LIN {X -0.215,Y -608.522,Z 1231.656,A 0.000,B 0.000,C 90.000,E1 154.152} C_DIS
LIN {X 0.197,Y -611.712,Z 1231.652,A 0.000,B 0.000,C 90.000,E1 153.332} C_DIS
LIN {X 0.064,Y -615.753,Z 1231.646,A 0.000,B 0.000,C 90.000,E1 152.308} C_DIS
LIN {X -0.293,Y -621.493,Z 1231.638,A 0.000,B 0.000,C 90.000,E1 150.795} C_DIS
LIN {X -0.001,Y -625.230,Z 1231.632,A 0.000,B 0.000,C 90.000,E1 149.744} C_DIS
LIN {X -0.198,Y -628.990,Z 1231.626,A 0.000,B 0.000,C 90.000,E1 148.742} C_DIS
LIN {X 0.009,Y -633.541,Z 1231.619,A 0.000,B 0.000,C 90.000,E1 147.454} C_DIS
LIN {X -0.240,Y -637.777,Z 1231.612,A 0.000,B 0.000,C 90.000,E1 146.215} C_DIS
LIN {X -0.421,Y -641.797,Z 1231.605,A 0.000,B 0.000,C 90.000,E1 144.975} C_DIS
LIN {X -0.172,Y -645.344,Z 1231.598,A 0.000,B 0.000,C 90.000,E1 143.703} C_DIS
LIN {X -0.235,Y -646.733,Z 1231.596,A 0.000,B 0.000,C 90.000,E1 143.210} C_DIS
LIN {X -0.024,Y -649.852,Z 1231.589,A 0.000,B 0.000,C 90.000,E1 141.949} C_DIS
LIN {X 0.287,Y -653.430,Z 1231.580,A 0.000,B 0.000,C 90.000,E1 140.436} C_DIS
LIN {X 0.118,Y -656.246,Z 1231.573,A 0.000,B 0.000,C 90.000,E1 139.218} C_DIS
LIN {X -0.055,Y -660.199,Z 1231.564,A 0.000,B 0.000,C 90.000,E1 137.514} C_DIS
LIN {X -0.154,Y -664.675,Z 1231.553,A 0.000,B 0.000,C 90.000,E1 135.567} C_DIS
LIN {X -0.165,Y -668.917,Z 1231.544,A 0.000,B 0.000,C 90.000,E1 133.866} C_DIS
LIN {X -0.055,Y -673.267,Z 1231.534,A 0.000,B 0.000,C 90.000,E1 132.162} C_DIS
LIN {X 0.130,Y -676.933,Z 1231.526,A 0.000,B 0.000,C 90.000,E1 130.701} C_DIS
LIN {X -0.089,Y -680.001,Z 1231.520,A 0.000,B 0.000,C 90.000,E1 129.519} C_DIS
LIN {X -0.223,Y -683.658,Z 1231.512,A 0.000,B 0.000,C 90.000,E1 128.096} C_DIS
LIN {X -0.178,Y -687.277,Z 1231.504,A 0.000,B 0.000,C 90.000,E1 126.664} C_DIS
LIN {X -0.296,Y -689.544,Z 1231.498,A 0.000,B 0.000,C 90.000,E1 125.724} C_DIS
LIN {X 0.024,Y -692.770,Z 1231.490,A 0.000,B 0.000,C 90.000,E1 124.278} C_DIS
LIN {X 0.183,Y -695.394,Z 1231.484,A 0.000,B 0.000,C 90.000,E1 123.086} C_DIS
LIN {X 0.339,Y -697.341,Z 1231.479,A 0.000,B 0.000,C 90.000,E1 122.133} C_DIS
LIN {X -0.187,Y -699.644,Z 1231.472,A 0.000,B 0.000,C 90.000,E1 121.003} C_DIS
LIN {X 0.015,Y -701.391,Z 1231.467,A 0.000,B 0.000,C 90.000,E1 120.050} C_DIS
LIN {X -0.121,Y -703.044,Z 1231.462,A 0.000,B 0.000,C 90.000,E1 119.127} C_DIS
LIN {X 0.099,Y -704.093,Z 1231.458,A 0.000,B 0.000,C 90.000,E1 118.409} C_DIS
LIN {X 0.000,Y -704.953,Z 1231.454,A 0.000,B 0.000,C 90.000,E1 117.719} C_DIS
LIN {X 0.241,Y -705.565,Z 1231.450,A 0.000,B 0.000,C 90.000,E1 117.001} C_DIS
LIN {X 0.170,Y -706.015,Z 1231.446,A 0.000,B 0.000,C 90.000,E1 116.309} C_DIS
LIN {X 0.413,Y -706.169,Z 1231.442,A 0.000,B 0.000,C 90.000,E1 115.591} C_DIS
LIN {X 0.058,Y -706.120,Z 1231.440,A 0.000,B 0.000,C 90.000,E1 115.155} C_DIS
LIN {X 0.001,Y -705.807,Z 1231.437,A 0.000,B 0.000,C 90.000,E1 114.695} C_DIS
LIN {X -0.003,Y -705.533,Z 1231.436,A 0.000,B 0.000,C 90.000,E1 114.463} C_DIS
LIN {X -0.069,Y -704.719,Z 1231.433,A 0.000,B 0.000,C 90.000,E1 114.003} C_DIS
LIN {X -0.069,Y -703.824,Z 1231.432,A 0.000,B 0.000,C 90.000,E1 113.770} C_DIS
LIN {X -0.429,Y -701.590,Z 1231.429,A 0.000,B 0.000,C 90.000,E1 113.334} C_DIS
LIN {X -0.291,Y -700.673,Z 1231.429,A 0.000,B 0.000,C 90.000,E1 113.206} C_DIS
LIN {X 0.148,Y -695.709,Z 1231.426,A 0.000,B 0.000,C 90.000,E1 112.717} C_DIS
LIN {X -0.315,Y -694.073,Z 1231.426,A 0.000,B 0.000,C 90.000,E1 112.642} C_DIS
LIN {X 0.049,Y -691.649,Z 1231.425,A 0.000,B 0.000,C 90.000,E1 112.514} C_DIS
LIN {X -0.259,Y -686.935,Z 1231.424,A 0.000,B 0.000,C 90.000,E1 112.386} C_DIS
LIN {X -0.290,Y -683.690,Z 1231.424,A 0.000,B 0.000,C 90.000,E1 112.333} C_DIS
LIN {X -0.124,Y -676.958,Z 1231.424,A 0.000,B 0.000,C 90.000,E1 112.280} C_DIS
LIN {X -0.162,Y -617.564,Z 1231.424,A 0.000,B 0.000,C 90.000,E1 112.280} C_DIS
LIN {X 0.169,Y -614.890,Z 1231.423,A 0.000,B 0.000,C 90.000,E1 112.099} C_DIS
LIN {X -0.080,Y -611.777,Z 1231.421,A 0.000,B 0.000,C 90.000,E1 111.844} C_DIS
LIN {X 0.070,Y -611.245,Z 1231.421,A 0.000,B 0.000,C 90.000,E1 111.770} C_DIS
LIN {X -0.103,Y -610.878,Z 1231.421,A 0.000,B 0.000,C 90.000,E1 111.716} C_DIS
LIN {X -0.008,Y -610.901,Z 1231.420,A 0.000,B 0.000,C 90.000,E1 111.535} C_DIS
LIN {X -0.055,Y -611.491,Z 1231.418,A 0.000,B 0.000,C 90.000,E1 111.280} C_DIS
LIN {X -0.324,Y -612.402,Z 1231.417,A 0.000,B 0.000,C 90.000,E1 111.046} C_DIS
LIN {X -0.008,Y -617.164,Z 1231.411,A 0.000,B 0.000,C 90.000,E1 109.993} C_DIS
LIN {X 0.052,Y -620.407,Z 1231.407,A 0.000,B 0.000,C 90.000,E1 109.214} C_DIS
LIN {X -0.211,Y -622.301,Z 1231.404,A 0.000,B 0.000,C 90.000,E1 108.725} C_DIS
LIN {X 0.129,Y -624.409,Z 1231.401,A 0.000,B 0.000,C 90.000,E1 108.181} C_DIS
LIN {X -0.348,Y -631.904,Z 1231.391,A 0.000,B 0.000,C 90.000,E1 106.441} C_DIS
LIN {X 0.056,Y -634.072,Z 1231.388,A 0.000,B 0.000,C 90.000,E1 105.898} C_DIS
LIN {X 0.126,Y -636.956,Z 1231.384,A 0.000,B 0.000,C 90.000,E1 105.134} C_DIS
LIN {X -0.226,Y -639.190,Z 1231.380,A 0.000,B 0.000,C 90.000,E1 104.411} C_DIS
LIN {X 0.061,Y -640.555,Z 1231.377,A 0.000,B 0.000,C 90.000,E1 103.883} C_DIS
LIN {X 0.045,Y -642.355,Z 1231.372,A 0.000,B 0.000,C 90.000,E1 102.883} C_DIS
LIN {X -0.111,Y -642.699,Z 1231.370,A 0.000,B 0.000,C 90.000,E1 102.647} C_DIS
LIN {X 0.206,Y -642.910,Z 1231.367,A 0.000,B 0.000,C 90.000,E1 102.119} C_DIS
LIN {X 0.240,Y -642.508,Z 1231.363,A 0.000,B 0.000,C 90.000,E1 101.366} C_DIS
LIN {X -0.072,Y -641.928,Z 1231.361,A 0.000,B 0.000,C 90.000,E1 100.894} C_DIS
LIN {X 0.238,Y -640.857,Z 1231.358,A 0.000,B 0.000,C 90.000,E1 100.366} C_DIS
LIN {X -0.202,Y -639.493,Z 1231.355,A 0.000,B 0.000,C 90.000,E1 99.905} C_DIS
LIN {X 0.088,Y -637.800,Z 1231.352,A 0.000,B 0.000,C 90.000,E1 99.378} C_DIS
LIN {X 0.263,Y -635.771,Z 1231.349,A 0.000,B 0.000,C 90.000,E1 98.859} C_DIS
LIN {X 0.080,Y -634.653,Z 1231.348,A 0.000,B 0.000,C 90.000,E1 98.624} C_DIS
LIN {X 0.091,Y -631.158,Z 1231.344,A 0.000,B 0.000,C 90.000,E1 97.992} C_DIS
LIN {X 0.224,Y -627.938,Z 1231.342,A 0.000,B 0.000,C 90.000,E1 97.473} C_DIS
LIN {X -0.134,Y -625.212,Z 1231.340,A 0.000,B 0.000,C 90.000,E1 97.125} C_DIS
LIN {X -0.123,Y -619.843,Z 1231.336,A 0.000,B 0.000,C 90.000,E1 96.486} C_DIS
LIN {X 0.026,Y -616.006,Z 1231.334,A 0.000,B 0.000,C 90.000,E1 96.087} C_DIS
LIN {X -0.273,Y -610.789,Z 1231.331,A 0.000,B 0.000,C 90.000,E1 95.625} C_DIS
LIN {X 0.251,Y -607.948,Z 1231.330,A 0.000,B 0.000,C 90.000,E1 95.334} C_DIS
LIN {X -0.273,Y -601.860,Z 1231.327,A 0.000,B 0.000,C 90.000,E1 94.935} C_DIS
LIN {X 0.266,Y -595.811,Z 1231.325,A 0.000,B 0.000,C 90.000,E1 94.473} C_DIS
LIN {X 0.137,Y -591.134,Z 1231.323,A 0.000,B 0.000,C 90.000,E1 94.188} C_DIS
LIN {X 0.120,Y -582.888,Z 1231.321,A 0.000,B 0.000,C 90.000,E1 93.726} C_DIS
LIN {X -0.057,Y -572.286,Z 1231.318,A 0.000,B 0.000,C 90.000,E1 93.269} C_DIS
LIN {X -0.105,Y -566.701,Z 1231.317,A 0.000,B 0.000,C 90.000,E1 92.980} C_DIS
LIN {X -0.264,Y -566.416,Z 1231.316,A 0.000,B 0.000,C 90.000,E1 92.980} C_DIS
LIN {X 0.250,Y -566.379,Z 1231.316,A 0.000,B 0.000,C 90.000,E1 92.922} C_DIS
LIN {X -0.100,Y -566.232,Z 1231.316,A 0.000,B 0.000,C 90.000,E1 92.808} C_DIS
LIN {X 0.014,Y -565.736,Z 1231.314,A 0.000,B 0.000,C 90.000,E1 92.522} C_DIS
LIN {X -0.213,Y -565.373,Z 1231.313,A 0.000,B 0.000,C 90.000,E1 92.407} C_DIS
LIN {X 0.239,Y -565.345,Z 1231.311,A 0.000,B 0.000,C 90.000,E1 91.949} C_DIS
LIN {X 0.154,Y -566.958,Z 1231.297,A 0.000,B 0.000,C 90.000,E1 89.484} C_DIS
LIN {X -0.249,Y -568.116,Z 1231.288,A 0.000,B 0.000,C 90.000,E1 87.879} C_DIS
LIN {X 0.099,Y -569.642,Z 1231.277,A 0.000,B 0.000,C 90.000,E1 85.927} C_DIS
LIN {X 0.081,Y -571.596,Z 1231.265,A 0.000,B 0.000,C 90.000,E1 83.742} C_DIS
LIN {X -0.149,Y -573.187,Z 1231.256,A 0.000,B 0.000,C 90.000,E1 82.129} C_DIS
LIN {X 0.179,Y -574.429,Z 1231.249,A 0.000,B 0.000,C 90.000,E1 80.735} C_DIS
LIN {X -0.033,Y -575.456,Z 1231.241,A 0.000,B 0.000,C 90.000,E1 79.398} C_DIS
LIN {X 0.305,Y -576.731,Z 1231.231,A 0.000,B 0.000,C 90.000,E1 77.465} C_DIS
LIN {X 0.030,Y -577.406,Z 1231.225,A 0.000,B 0.000,C 90.000,E1 76.408} C_DIS
LIN {X 0.114,Y -578.199,Z 1231.217,A 0.000,B 0.000,C 90.000,E1 75.046} C_DIS
LIN {X 0.026,Y -579.070,Z 1231.208,A 0.000,B 0.000,C 90.000,E1 73.433} C_DIS
LIN {X 0.125,Y -579.827,Z 1231.201,A 0.000,B 0.000,C 90.000,E1 72.072} C_DIS
LIN {X -0.122,Y -580.862,Z 1231.192,A 0.000,B 0.000,C 90.000,E1 70.477} C_DIS
LIN {X 0.164,Y -582.757,Z 1231.175,A 0.000,B 0.000,C 90.000,E1 67.486} C_DIS
LIN {X -0.066,Y -583.664,Z 1231.169,A 0.000,B 0.000,C 90.000,E1 66.433} C_DIS
LIN {X 0.231,Y -585.122,Z 1231.160,A 0.000,B 0.000,C 90.000,E1 64.793} C_DIS
LIN {X 0.061,Y -587.057,Z 1231.148,A 0.000,B 0.000,C 90.000,E1 62.666} C_DIS
LIN {X 0.284,Y -588.446,Z 1231.141,A 0.000,B 0.000,C 90.000,E1 61.307} C_DIS
LIN {X 0.012,Y -589.829,Z 1231.133,A 0.000,B 0.000,C 90.000,E1 59.999} C_DIS
LIN {X 0.055,Y -591.209,Z 1231.126,A 0.000,B 0.000,C 90.000,E1 58.663} C_DIS
LIN {X 0.120,Y -592.435,Z 1231.119,A 0.000,B 0.000,C 90.000,E1 57.327} C_DIS
LIN {X -0.189,Y -593.426,Z 1231.113,A 0.000,B 0.000,C 90.000,E1 56.294} C_DIS
LIN {X -0.267,Y -594.547,Z 1231.105,A 0.000,B 0.000,C 90.000,E1 54.975} C_DIS
LIN {X 0.021,Y -595.606,Z 1231.098,A 0.000,B 0.000,C 90.000,E1 53.623} C_DIS
LIN {X -0.289,Y -597.231,Z 1231.086,A 0.000,B 0.000,C 90.000,E1 51.537} C_DIS
LIN {X -0.058,Y -597.783,Z 1231.082,A 0.000,B 0.000,C 90.000,E1 50.723} C_DIS
LIN {X -0.026,Y -598.759,Z 1231.070,A 0.000,B 0.000,C 90.000,E1 48.609} C_DIS
LIN {X -0.004,Y -599.228,Z 1231.064,A 0.000,B 0.000,C 90.000,E1 47.553} C_DIS
LIN {X 0.209,Y -599.506,Z 1231.057,A 0.000,B 0.000,C 90.000,E1 46.215} C_DIS
LIN {X 0.210,Y -599.574,Z 1231.051,A 0.000,B 0.000,C 90.000,E1 45.162} C_DIS
LIN {X 0.000,Y -599.392,Z 1231.044,A 0.000,B 0.000,C 90.000,E1 43.866} C_DIS
LIN {X -0.203,Y -599.215,Z 1231.039,A 0.000,B 0.000,C 90.000,E1 43.095} C_DIS
LIN {X 0.000,Y -598.876,Z 1231.035,A 0.000,B 0.000,C 90.000,E1 42.285} C_DIS
LIN {X -0.200,Y -598.172,Z 1231.028,A 0.000,B 0.000,C 90.000,E1 40.987} C_DIS
LIN {X 0.044,Y -597.530,Z 1231.020,A 0.000,B 0.000,C 90.000,E1 39.644} C_DIS
LIN {X 0.042,Y -596.778,Z 1231.014,A 0.000,B 0.000,C 90.000,E1 38.588} C_DIS
LIN {X -0.104,Y -595.974,Z 1231.010,A 0.000,B 0.000,C 90.000,E1 37.810} C_DIS
LIN {X -0.024,Y -594.803,Z 1231.004,A 0.000,B 0.000,C 90.000,E1 36.744} C_DIS
LIN {X 0.169,Y -593.779,Z 1231.000,A 0.000,B 0.000,C 90.000,E1 35.931} C_DIS
LIN {X -0.128,Y -592.057,Z 1230.994,A 0.000,B 0.000,C 90.000,E1 34.898} C_DIS
LIN {X 0.173,Y -590.544,Z 1230.989,A 0.000,B 0.000,C 90.000,E1 34.072} C_DIS
LIN {X -0.035,Y -588.860,Z 1230.985,A 0.000,B 0.000,C 90.000,E1 33.293} C_DIS
LIN {X -0.090,Y -586.871,Z 1230.981,A 0.000,B 0.000,C 90.000,E1 32.498} C_DIS
LIN {X -0.029,Y -585.376,Z 1230.978,A 0.000,B 0.000,C 90.000,E1 31.957} C_DIS
LIN {X 0.060,Y -581.844,Z 1230.972,A 0.000,B 0.000,C 90.000,E1 30.875} C_DIS
LIN {X -0.057,Y -578.700,Z 1230.967,A 0.000,B 0.000,C 90.000,E1 30.079} C_DIS
LIN {X -0.131,Y -575.752,Z 1230.963,A 0.000,B 0.000,C 90.000,E1 29.411} C_DIS
LIN {X 0.103,Y -571.104,Z 1230.958,A 0.000,B 0.000,C 90.000,E1 28.437} C_DIS
LIN {X -0.227,Y -565.810,Z 1230.953,A 0.000,B 0.000,C 90.000,E1 27.513} C_DIS
LIN {X 0.069,Y -561.668,Z 1230.949,A 0.000,B 0.000,C 90.000,E1 26.796} C_DIS
LIN {X -0.137,Y -555.267,Z 1230.944,A 0.000,B 0.000,C 90.000,E1 25.848} C_DIS
LIN {X -0.182,Y -550.305,Z 1230.940,A 0.000,B 0.000,C 90.000,E1 25.155} C_DIS
LIN {X 0.104,Y -543.551,Z 1230.935,A 0.000,B 0.000,C 90.000,E1 24.283} C_DIS
LIN {X -0.178,Y -536.321,Z 1230.930,A 0.000,B 0.000,C 90.000,E1 23.462} C_DIS
LIN {X -0.243,Y -531.252,Z 1230.927,A 0.000,B 0.000,C 90.000,E1 22.898} C_DIS
LIN {X 0.041,Y -523.432,Z 1230.922,A 0.000,B 0.000,C 90.000,E1 22.025} C_DIS
LIN {X 0.086,Y -518.116,Z 1230.919,A 0.000,B 0.000,C 90.000,E1 21.461} C_DIS
LIN {X 0.164,Y -508.565,Z 1230.914,A 0.000,B 0.000,C 90.000,E1 20.482} C_DIS
LIN {X -0.201,Y -498.708,Z 1230.909,A 0.000,B 0.000,C 90.000,E1 19.577} C_DIS
LIN {X 0.190,Y -490.108,Z 1230.904,A 0.000,B 0.000,C 90.000,E1 18.725} C_DIS
LIN {X 0.240,Y -480.107,Z 1230.899,A 0.000,B 0.000,C 90.000,E1 17.819} C_DIS
LIN {X 0.020,Y -466.906,Z 1230.893,A 0.000,B 0.000,C 90.000,E1 16.677} C_DIS
LIN {X 0.134,Y -450.553,Z 1230.885,A 0.000,B 0.000,C 90.000,E1 15.190} C_DIS
LIN {X -0.149,Y -431.722,Z 1230.874,A 0.000,B 0.000,C 90.000,E1 13.411} C_DIS
LIN {X -0.016,Y -414.674,Z 1230.864,A 0.000,B 0.000,C 90.000,E1 11.591} C_DIS
LIN {X 0.035,Y -400.676,Z 1230.855,A 0.000,B 0.000,C 90.000,E1 9.962} C_DIS
LIN {X 0.040,Y -396.618,Z 1230.852,A 0.000,B 0.000,C 90.000,E1 9.378} C_DIS
LIN {X -0.002,Y -395.476,Z 1230.851,A 0.000,B 0.000,C 90.000,E1 9.208} C_DIS
LIN {X -0.091,Y -394.124,Z 1230.849,A 0.000,B 0.000,C 90.000,E1 8.859} C_DIS
LIN {X -0.120,Y -394.118,Z 1230.849,A 0.000,B 0.000,C 90.000,E1 8.859} C_DIS
LIN {X -0.126,Y -394.090,Z 1230.848,A 0.000,B 0.000,C 90.000,E1 8.681} C_DIS
LIN {X -0.164,Y -394.095,Z 1230.848,A 0.000,B 0.000,C 90.000,E1 8.681} C_DIS
LIN {X 0.077,Y -396.818,Z 1230.845,A 0.000,B 0.000,C 90.000,E1 8.049} C_DIS
LIN {X 0.018,Y -400.484,Z 1230.843,A 0.000,B 0.000,C 90.000,E1 7.644} C_DIS
LIN {X 0.065,Y -407.645,Z 1230.839,A 0.000,B 0.000,C 90.000,E1 7.068} C_DIS
LIN {X -0.064,Y -414.167,Z 1230.837,A 0.000,B 0.000,C 90.000,E1 6.606} C_DIS
LIN {X -0.218,Y -420.667,Z 1230.834,A 0.000,B 0.000,C 90.000,E1 6.144} C_DIS
LIN {X 0.068,Y -423.501,Z 1230.833,A 0.000,B 0.000,C 90.000,E1 5.910} C_DIS
LIN {X -0.169,Y -434.411,Z 1230.828,A 0.000,B 0.000,C 90.000,E1 5.106} C_DIS
LIN {X 0.204,Y -448.610,Z 1230.822,A 0.000,B 0.000,C 90.000,E1 3.955} C_DIS
LIN {X -0.209,Y -459.626,Z 1230.817,A 0.000,B 0.000,C 90.000,E1 3.151} C_DIS
LIN {X -0.008,Y -467.146,Z 1230.814,A 0.000,B 0.000,C 90.000,E1 2.522} C_DIS
LIN {X 0.065,Y -473.129,Z 1230.811,A 0.000,B 0.000,C 90.000,E1 2.007} C_DIS
LIN {X -0.017,Y -478.963,Z 1230.808,A 0.000,B 0.000,C 90.000,E1 1.489} C_DIS
LIN {X -0.155,Y -484.492,Z 1230.805,A 0.000,B 0.000,C 90.000,E1 0.974} C_DIS
LIN {X 0.187,Y -491.248,Z 1230.801,A 0.000,B 0.000,C 90.000,E1 0.229} C_DIS
LIN {X -0.229,Y -497.810,Z 1230.797,A 0.000,B 0.000,C 90.000,E1 359.542} C_DIS
LIN {X 0.232,Y -503.893,Z 1230.793,A 0.000,B 0.000,C 90.000,E1 358.740} C_DIS
LIN {X 0.229,Y -509.539,Z 1230.789,A 0.000,B 0.000,C 90.000,E1 357.993} C_DIS
LIN {X -0.251,Y -514.703,Z 1230.785,A 0.000,B 0.000,C 90.000,E1 357.306} C_DIS
LIN {X 0.142,Y -518.609,Z 1230.782,A 0.000,B 0.000,C 90.000,E1 356.674} C_DIS
LIN {X -0.274,Y -523.122,Z 1230.778,A 0.000,B 0.000,C 90.000,E1 355.988} C_DIS
LIN {X -0.095,Y -527.203,Z 1230.774,A 0.000,B 0.000,C 90.000,E1 355.241} C_DIS
LIN {X -0.125,Y -530.223,Z 1230.770,A 0.000,B 0.000,C 90.000,E1 354.666} C_DIS
LIN {X 0.175,Y -533.700,Z 1230.766,A 0.000,B 0.000,C 90.000,E1 353.913} C_DIS
LIN {X 0.197,Y -536.253,Z 1230.763,A 0.000,B 0.000,C 90.000,E1 353.337} C_DIS
LIN {X 0.294,Y -539.745,Z 1230.758,A 0.000,B 0.000,C 90.000,E1 352.470} C_DIS
LIN {X -0.110,Y -542.932,Z 1230.754,A 0.000,B 0.000,C 90.000,E1 351.659} C_DIS
LIN {X 0.052,Y -545.792,Z 1230.749,A 0.000,B 0.000,C 90.000,E1 350.792} C_DIS
LIN {X 0.146,Y -547.586,Z 1230.746,A 0.000,B 0.000,C 90.000,E1 350.218} C_DIS
LIN {X -0.094,Y -549.966,Z 1230.741,A 0.000,B 0.000,C 90.000,E1 349.398} C_DIS
LIN {X -0.186,Y -552.951,Z 1230.735,A 0.000,B 0.000,C 90.000,E1 348.285} C_DIS
LIN {X 0.179,Y -555.021,Z 1230.730,A 0.000,B 0.000,C 90.000,E1 347.409} C_DIS
LIN {X 0.153,Y -557.506,Z 1230.724,A 0.000,B 0.000,C 90.000,E1 346.297} C_DIS
LIN {X -0.249,Y -559.814,Z 1230.718,A 0.000,B 0.000,C 90.000,E1 345.227} C_DIS
LIN {X 0.224,Y -562.343,Z 1230.710,A 0.000,B 0.000,C 90.000,E1 343.795} C_DIS
LIN {X -0.108,Y -564.102,Z 1230.704,A 0.000,B 0.000,C 90.000,E1 342.725} C_DIS
LIN {X 0.137,Y -565.293,Z 1230.699,A 0.000,B 0.000,C 90.000,E1 341.873} C_DIS
LIN {X 0.015,Y -566.668,Z 1230.693,A 0.000,B 0.000,C 90.000,E1 340.786} C_DIS
LIN {X 0.296,Y -567.424,Z 1230.689,A 0.000,B 0.000,C 90.000,E1 339.934} C_DIS
LIN {X 0.052,Y -568.003,Z 1230.684,A 0.000,B 0.000,C 90.000,E1 339.135} C_DIS
LIN {X 0.001,Y -568.239,Z 1230.681,A 0.000,B 0.000,C 90.000,E1 338.592} C_DIS
LIN {X -0.239,Y -568.354,Z 1230.677,A 0.000,B 0.000,C 90.000,E1 337.794} C_DIS
LIN {X -0.078,Y -568.251,Z 1230.673,A 0.000,B 0.000,C 90.000,E1 337.230} C_DIS
LIN {X 0.085,Y -568.003,Z 1230.670,A 0.000,B 0.000,C 90.000,E1 336.666} C_DIS
LIN {X 0.067,Y -567.323,Z 1230.666,A 0.000,B 0.000,C 90.000,E1 335.845} C_DIS
LIN {X -0.012,Y -566.721,Z 1230.663,A 0.000,B 0.000,C 90.000,E1 335.305} C_DIS
LIN {X 0.195,Y -565.461,Z 1230.658,A 0.000,B 0.000,C 90.000,E1 334.460} C_DIS
LIN {X 0.148,Y -563.925,Z 1230.654,A 0.000,B 0.000,C 90.000,E1 333.640} C_DIS
LIN {X 0.143,Y -561.227,Z 1230.648,A 0.000,B 0.000,C 90.000,E1 332.538} C_DIS
LIN {X -0.250,Y -559.742,Z 1230.645,A 0.000,B 0.000,C 90.000,E1 332.025} C_DIS
LIN {X -0.105,Y -556.742,Z 1230.640,A 0.000,B 0.000,C 90.000,E1 331.179} C_DIS
LIN {X 0.225,Y -554.373,Z 1230.637,A 0.000,B 0.000,C 90.000,E1 330.589} C_DIS
LIN {X 0.053,Y -551.812,Z 1230.634,A 0.000,B 0.000,C 90.000,E1 330.049} C_DIS
LIN {X 0.220,Y -548.265,Z 1230.630,A 0.000,B 0.000,C 90.000,E1 329.331} C_DIS
LIN {X -0.117,Y -543.983,Z 1230.626,A 0.000,B 0.000,C 90.000,E1 328.663} C_DIS
LIN {X -0.031,Y -539.296,Z 1230.622,A 0.000,B 0.000,C 90.000,E1 327.946} C_DIS
LIN {X -0.015,Y -535.303,Z 1230.619,A 0.000,B 0.000,C 90.000,E1 327.375} C_DIS
LIN {X 0.119,Y -528.921,Z 1230.614,A 0.000,B 0.000,C 90.000,E1 326.501} C_DIS
LIN {X 0.074,Y -517.700,Z 1230.606,A 0.000,B 0.000,C 90.000,E1 325.055} C_DIS
LIN {X -0.049,Y -513.713,Z 1230.603,A 0.000,B 0.000,C 90.000,E1 324.482} C_DIS
LIN {X 0.066,Y -512.792,Z 1230.602,A 0.000,B 0.000,C 90.000,E1 324.322} C_DIS
LIN {X 0.105,Y -510.374,Z 1230.599,A 0.000,B 0.000,C 90.000,E1 323.829} C_DIS
LIN {X -0.263,Y -508.097,Z 1230.595,A 0.000,B 0.000,C 90.000,E1 323.130} C_DIS
LIN {X 0.059,Y -507.015,Z 1230.591,A 0.000,B 0.000,C 90.000,E1 322.351} C_DIS
LIN {X 0.075,Y -506.370,Z 1230.586,A 0.000,B 0.000,C 90.000,E1 321.457} C_DIS
LIN {X 0.089,Y -506.452,Z 1230.581,A 0.000,B 0.000,C 90.000,E1 320.561} C_DIS
LIN {X 0.247,Y -507.707,Z 1230.568,A 0.000,B 0.000,C 90.000,E1 318.162} C_DIS
LIN {X 0.128,Y -508.323,Z 1230.561,A 0.000,B 0.000,C 90.000,E1 316.986} C_DIS
LIN {X 0.259,Y -508.949,Z 1230.553,A 0.000,B 0.000,C 90.000,E1 315.486} C_DIS
LIN {X 0.035,Y -509.489,Z 1230.545,A 0.000,B 0.000,C 90.000,E1 314.028} C_DIS
LIN {X -0.050,Y -510.330,Z 1230.533,A 0.000,B 0.000,C 90.000,E1 311.962} C_DIS
LIN {X -0.091,Y -510.828,Z 1230.527,A 0.000,B 0.000,C 90.000,E1 310.782} C_DIS
LIN {X 0.126,Y -511.359,Z 1230.518,A 0.000,B 0.000,C 90.000,E1 309.277} C_DIS
LIN {X -0.056,Y -511.923,Z 1230.508,A 0.000,B 0.000,C 90.000,E1 307.523} C_DIS
LIN {X 0.176,Y -512.442,Z 1230.499,A 0.000,B 0.000,C 90.000,E1 305.724} C_DIS
LIN {X -0.180,Y -512.957,Z 1230.489,A 0.000,B 0.000,C 90.000,E1 303.992} C_DIS
LIN {X -0.096,Y -513.368,Z 1230.479,A 0.000,B 0.000,C 90.000,E1 302.212} C_DIS
LIN {X -0.280,Y -513.541,Z 1230.469,A 0.000,B 0.000,C 90.000,E1 300.463} C_DIS
LIN {X 0.072,Y -513.648,Z 1230.461,A 0.000,B 0.000,C 90.000,E1 298.949} C_DIS
LIN {X 0.072,Y -513.713,Z 1230.451,A 0.000,B 0.000,C 90.000,E1 297.180} C_DIS
LIN {X -0.282,Y -513.780,Z 1230.440,A 0.000,B 0.000,C 90.000,E1 295.155} C_DIS
LIN {X 0.067,Y -513.926,Z 1230.431,A 0.000,B 0.000,C 90.000,E1 293.643} C_DIS
LIN {X 0.211,Y -513.828,Z 1230.423,A 0.000,B 0.000,C 90.000,E1 292.153} C_DIS
LIN {X 0.104,Y -513.543,Z 1230.418,A 0.000,B 0.000,C 90.000,E1 291.280} C_DIS
LIN {X 0.046,Y -512.929,Z 1230.410,A 0.000,B 0.000,C 90.000,E1 289.812} C_DIS
LIN {X -0.194,Y -512.276,Z 1230.402,A 0.000,B 0.000,C 90.000,E1 288.362} C_DIS
LIN {X 0.105,Y -511.343,Z 1230.391,A 0.000,B 0.000,C 90.000,E1 286.260} C_DIS
LIN {X 0.217,Y -510.821,Z 1230.384,A 0.000,B 0.000,C 90.000,E1 285.064} C_DIS
LIN {X 0.069,Y -509.603,Z 1230.372,A 0.000,B 0.000,C 90.000,E1 283.008} C_DIS
LIN {X -0.110,Y -508.133,Z 1230.361,A 0.000,B 0.000,C 90.000,E1 280.950} C_DIS
LIN {X -0.077,Y -506.417,Z 1230.348,A 0.000,B 0.000,C 90.000,E1 278.568} C_DIS
LIN {X 0.201,Y -504.823,Z 1230.333,A 0.000,B 0.000,C 90.000,E1 275.853} C_DIS
LIN {X 0.013,Y -503.641,Z 1230.321,A 0.000,B 0.000,C 90.000,E1 273.784} C_DIS
LIN {X -0.144,Y -502.551,Z 1230.311,A 0.000,B 0.000,C 90.000,E1 272.007} C_DIS
LIN {X -0.090,Y -501.610,Z 1230.304,A 0.000,B 0.000,C 90.000,E1 270.802} C_DIS
LIN {X 0.200,Y -500.447,Z 1230.294,A 0.000,B 0.000,C 90.000,E1 268.969} C_DIS
LIN {X -0.030,Y -499.371,Z 1230.284,A 0.000,B 0.000,C 90.000,E1 267.192} C_DIS
LIN {X -0.025,Y -498.705,Z 1230.278,A 0.000,B 0.000,C 90.000,E1 265.988} C_DIS
LIN {X 0.005,Y -498.005,Z 1230.271,A 0.000,B 0.000,C 90.000,E1 264.780} C_DIS
LIN {X -0.066,Y -496.871,Z 1230.263,A 0.000,B 0.000,C 90.000,E1 263.280} C_DIS
LIN {X -0.160,Y -495.514,Z 1230.254,A 0.000,B 0.000,C 90.000,E1 261.781} C_DIS
LIN {X -0.216,Y -494.107,Z 1230.246,A 0.000,B 0.000,C 90.000,E1 260.274} C_DIS
LIN {X 0.074,Y -492.037,Z 1230.232,A 0.000,B 0.000,C 90.000,E1 257.813} C_DIS
LIN {X -0.162,Y -490.163,Z 1230.217,A 0.000,B 0.000,C 90.000,E1 255.102} C_DIS
LIN {X -0.090,Y -488.675,Z 1230.204,A 0.000,B 0.000,C 90.000,E1 252.653} C_DIS
LIN {X 0.154,Y -488.082,Z 1230.197,A 0.000,B 0.000,C 90.000,E1 251.402} C_DIS
LIN {X 0.114,Y -487.177,Z 1230.187,A 0.000,B 0.000,C 90.000,E1 249.571} C_DIS
LIN {X 0.033,Y -486.345,Z 1230.178,A 0.000,B 0.000,C 90.000,E1 248.050} C_DIS
LIN {X 0.283,Y -485.627,Z 1230.171,A 0.000,B 0.000,C 90.000,E1 246.794} C_DIS
LIN {X 0.105,Y -484.172,Z 1230.161,A 0.000,B 0.000,C 90.000,E1 244.973} C_DIS
LIN {X -0.127,Y -482.180,Z 1230.147,A 0.000,B 0.000,C 90.000,E1 242.538} C_DIS
LIN {X 0.057,Y -480.746,Z 1230.139,A 0.000,B 0.000,C 90.000,E1 240.973} C_DIS
LIN {X -0.001,Y -479.448,Z 1230.132,A 0.000,B 0.000,C 90.000,E1 239.744} C_DIS
LIN {X -0.055,Y -477.789,Z 1230.123,A 0.000,B 0.000,C 90.000,E1 238.201} C_DIS
LIN {X 0.117,Y -476.146,Z 1230.115,A 0.000,B 0.000,C 90.000,E1 236.628} C_DIS
LIN {X -0.138,Y -474.468,Z 1230.106,A 0.000,B 0.000,C 90.000,E1 235.102} C_DIS
LIN {X 0.018,Y -472.560,Z 1230.096,A 0.000,B 0.000,C 90.000,E1 233.210} C_DIS
LIN {X 0.098,Y -470.430,Z 1230.083,A 0.000,B 0.000,C 90.000,E1 231.009} C_DIS
LIN {X -0.239,Y -468.559,Z 1230.071,A 0.000,B 0.000,C 90.000,E1 228.852} C_DIS
LIN {X -0.018,Y -466.718,Z 1230.059,A 0.000,B 0.000,C 90.000,E1 226.620} C_DIS
LIN {X -0.086,Y -463.920,Z 1230.026,A 0.000,B 0.000,C 90.000,E1 220.620} C_DIS
LIN {X 0.196,Y -465.253,Z 1229.998,A 0.000,B 0.000,C 90.000,E1 215.518} C_DIS
LIN {X -0.141,Y -467.489,Z 1229.978,A 0.000,B 0.000,C 90.000,E1 212.084} C_DIS
LIN {X 0.240,Y -469.027,Z 1229.969,A 0.000,B 0.000,C 90.000,E1 210.463} C_DIS
LIN {X 0.205,Y -472.106,Z 1229.954,A 0.000,B 0.000,C 90.000,E1 207.641} C_DIS
LIN {X 0.117,Y -474.826,Z 1229.942,A 0.000,B 0.000,C 90.000,E1 205.463} C_DIS
LIN {X -0.187,Y -480.394,Z 1229.921,A 0.000,B 0.000,C 90.000,E1 201.770} C_DIS
LIN {X -0.037,Y -487.434,Z 1229.900,A 0.000,B 0.000,C 90.000,E1 198.055} C_DIS
LIN {X -0.076,Y -494.447,Z 1229.883,A 0.000,B 0.000,C 90.000,E1 195.009} C_DIS
LIN {X 0.089,Y -499.058,Z 1229.873,A 0.000,B 0.000,C 90.000,E1 193.175} C_DIS
LIN {X 0.206,Y -502.995,Z 1229.865,A 0.000,B 0.000,C 90.000,E1 191.658} C_DIS
LIN {X -0.239,Y -509.571,Z 1229.852,A 0.000,B 0.000,C 90.000,E1 189.321} C_DIS
LIN {X 0.027,Y -512.993,Z 1229.845,A 0.000,B 0.000,C 90.000,E1 188.106} C_DIS
LIN {X -0.255,Y -517.113,Z 1229.837,A 0.000,B 0.000,C 90.000,E1 186.663} C_DIS
LIN {X -0.007,Y -522.074,Z 1229.827,A 0.000,B 0.000,C 90.000,E1 184.878} C_DIS
LIN {X -0.182,Y -526.964,Z 1229.818,A 0.000,B 0.000,C 90.000,E1 183.151} C_DIS
LIN {X 0.227,Y -531.084,Z 1229.809,A 0.000,B 0.000,C 90.000,E1 181.661} C_DIS
LIN {X 0.174,Y -535.054,Z 1229.801,A 0.000,B 0.000,C 90.000,E1 180.229} C_DIS
LIN {X 0.187,Y -538.261,Z 1229.795,A 0.000,B 0.000,C 90.000,E1 179.083} C_DIS
LIN {X -0.263,Y -542.070,Z 1229.787,A 0.000,B 0.000,C 90.000,E1 177.707} C_DIS
LIN {X -0.134,Y -544.990,Z 1229.781,A 0.000,B 0.000,C 90.000,E1 176.560} C_DIS
LIN {X 0.154,Y -549.250,Z 1229.771,A 0.000,B 0.000,C 90.000,E1 174.837} C_DIS
LIN {X -0.014,Y -552.585,Z 1229.764,A 0.000,B 0.000,C 90.000,E1 173.451} C_DIS
LIN {X -0.071,Y -556.522,Z 1229.754,A 0.000,B 0.000,C 90.000,E1 171.781} C_DIS
LIN {X -0.033,Y -559.677,Z 1229.747,A 0.000,B 0.000,C 90.000,E1 170.387} C_DIS
LIN {X -0.095,Y -562.216,Z 1229.740,A 0.000,B 0.000,C 90.000,E1 169.285} C_DIS
LIN {X -0.241,Y -565.900,Z 1229.731,A 0.000,B 0.000,C 90.000,E1 167.645} C_DIS
LIN {X -0.176,Y -569.694,Z 1229.722,A 0.000,B 0.000,C 90.000,E1 165.992} C_DIS
LIN {X 0.160,Y -574.358,Z 1229.712,A 0.000,B 0.000,C 90.000,E1 164.047} C_DIS
LIN {X -0.051,Y -584.477,Z 1229.692,A 0.000,B 0.000,C 90.000,E1 160.550} C_DIS
LIN {X 0.051,Y -591.207,Z 1229.682,A 0.000,B 0.000,C 90.000,E1 158.666} C_DIS
LIN {X 0.209,Y -598.760,Z 1229.671,A 0.000,B 0.000,C 90.000,E1 156.794} C_DIS
LIN {X 0.072,Y -605.179,Z 1229.662,A 0.000,B 0.000,C 90.000,E1 155.229} C_DIS
LIN {X -0.096,Y -608.360,Z 1229.658,A 0.000,B 0.000,C 90.000,E1 154.460} C_DIS
LIN {X 0.319,Y -611.537,Z 1229.654,A 0.000,B 0.000,C 90.000,E1 153.640} C_DIS
LIN {X 0.166,Y -616.497,Z 1229.647,A 0.000,B 0.000,C 90.000,E1 152.359} C_DIS
LIN {X -0.168,Y -622.134,Z 1229.638,A 0.000,B 0.000,C 90.000,E1 150.845} C_DIS
LIN {X -0.176,Y -624.926,Z 1229.634,A 0.000,B 0.000,C 90.000,E1 150.078} C_DIS
LIN {X -0.044,Y -629.488,Z 1229.627,A 0.000,B 0.000,C 90.000,E1 148.791} C_DIS
LIN {X -0.161,Y -633.978,Z 1229.620,A 0.000,B 0.000,C 90.000,E1 147.533} C_DIS
LIN {X -0.408,Y -638.136,Z 1229.613,A 0.000,B 0.000,C 90.000,E1 146.294} C_DIS
LIN {X 0.306,Y -642.018,Z 1229.606,A 0.000,B 0.000,C 90.000,E1 144.975} C_DIS
LIN {X 0.043,Y -645.552,Z 1229.599,A 0.000,B 0.000,C 90.000,E1 143.749} C_DIS
LIN {X 0.021,Y -647.469,Z 1229.594,A 0.000,B 0.000,C 90.000,E1 143.004} C_DIS
LIN {X -0.194,Y -649.927,Z 1229.589,A 0.000,B 0.000,C 90.000,E1 142.029} C_DIS
LIN {X 0.061,Y -654.032,Z 1229.579,A 0.000,B 0.000,C 90.000,E1 140.275} C_DIS
LIN {X -0.055,Y -656.239,Z 1229.574,A 0.000,B 0.000,C 90.000,E1 139.299} C_DIS
LIN {X 0.256,Y -660.162,Z 1229.564,A 0.000,B 0.000,C 90.000,E1 137.553} C_DIS
LIN {X -0.334,Y -664.608,Z 1229.553,A 0.000,B 0.000,C 90.000,E1 135.648} C_DIS
LIN {X -0.351,Y -668.206,Z 1229.545,A 0.000,B 0.000,C 90.000,E1 134.190} C_DIS
LIN {X 0.213,Y -673.156,Z 1229.535,A 0.000,B 0.000,C 90.000,E1 132.204} C_DIS
LIN {X -0.056,Y -676.797,Z 1229.527,A 0.000,B 0.000,C 90.000,E1 130.782} C_DIS
LIN {X 0.157,Y -679.861,Z 1229.520,A 0.000,B 0.000,C 90.000,E1 129.564} C_DIS
LIN {X -0.412,Y -683.513,Z 1229.512,A 0.000,B 0.000,C 90.000,E1 128.177} C_DIS
LIN {X 0.044,Y -687.123,Z 1229.504,A 0.000,B 0.000,C 90.000,E1 126.710} C_DIS
LIN {X 0.075,Y -689.397,Z 1229.499,A 0.000,B 0.000,C 90.000,E1 125.758} C_DIS
LIN {X 0.226,Y -692.635,Z 1229.491,A 0.000,B 0.000,C 90.000,E1 124.326} C_DIS
LIN {X -0.005,Y -695.261,Z 1229.484,A 0.000,B 0.000,C 90.000,E1 123.166} C_DIS
LIN {X 0.152,Y -697.251,Z 1229.479,A 0.000,B 0.000,C 90.000,E1 122.212} C_DIS
LIN {X -0.010,Y -699.559,Z 1229.473,A 0.000,B 0.000,C 90.000,E1 121.052} C_DIS
LIN {X -0.166,Y -701.324,Z 1229.467,A 0.000,B 0.000,C 90.000,E1 120.129} C_DIS
LIN {X -0.299,Y -702.995,Z 1229.462,A 0.000,B 0.000,C 90.000,E1 119.205} C_DIS
LIN {X 0.206,Y -704.401,Z 1229.457,A 0.000,B 0.000,C 90.000,E1 118.231} C_DIS
LIN {X -0.182,Y -705.217,Z 1229.453,A 0.000,B 0.000,C 90.000,E1 117.564} C_DIS
LIN {X 0.026,Y -705.910,Z 1229.448,A 0.000,B 0.000,C 90.000,E1 116.616} C_DIS
LIN {X -0.040,Y -706.211,Z 1229.444,A 0.000,B 0.000,C 90.000,E1 115.924} C_DIS
LIN {X -0.091,Y -706.228,Z 1229.442,A 0.000,B 0.000,C 90.000,E1 115.463} C_DIS
LIN {X -0.153,Y -705.938,Z 1229.438,A 0.000,B 0.000,C 90.000,E1 114.771} C_DIS
LIN {X 0.138,Y -705.746,Z 1229.436,A 0.000,B 0.000,C 90.000,E1 114.515} C_DIS
LIN {X -0.217,Y -704.889,Z 1229.434,A 0.000,B 0.000,C 90.000,E1 114.079} C_DIS
LIN {X 0.070,Y -704.198,Z 1229.432,A 0.000,B 0.000,C 90.000,E1 113.823} C_DIS
LIN {X -0.292,Y -702.056,Z 1229.430,A 0.000,B 0.000,C 90.000,E1 113.387} C_DIS
LIN {X -0.153,Y -701.329,Z 1229.429,A 0.000,B 0.000,C 90.000,E1 113.259} C_DIS
LIN {X -0.016,Y -700.243,Z 1229.429,A 0.000,B 0.000,C 90.000,E1 113.131} C_DIS
LIN {X -0.196,Y -695.069,Z 1229.426,A 0.000,B 0.000,C 90.000,E1 112.695} C_DIS
LIN {X -0.241,Y -693.101,Z 1229.425,A 0.000,B 0.000,C 90.000,E1 112.589} C_DIS
LIN {X 0.137,Y -686.247,Z 1229.424,A 0.000,B 0.000,C 90.000,E1 112.333} C_DIS
LIN {X -0.115,Y -685.237,Z 1229.424,A 0.000,B 0.000,C 90.000,E1 112.333} C_DIS
LIN {X -0.056,Y -677.689,Z 1229.424,A 0.000,B 0.000,C 90.000,E1 112.280} C_DIS
LIN {X -0.103,Y -616.835,Z 1229.424,A 0.000,B 0.000,C 90.000,E1 112.280} C_DIS
LIN {X -0.189,Y -613.104,Z 1229.423,A 0.000,B 0.000,C 90.000,E1 112.078} C_DIS
LIN {X -0.146,Y -610.558,Z 1229.421,A 0.000,B 0.000,C 90.000,E1 111.844} C_DIS
LIN {X -0.059,Y -609.483,Z 1229.420,A 0.000,B 0.000,C 90.000,E1 111.663} C_DIS
LIN {X -0.102,Y -609.486,Z 1229.420,A 0.000,B 0.000,C 90.000,E1 111.663} C_DIS
LIN {X 0.342,Y -609.739,Z 1229.418,A 0.000,B 0.000,C 90.000,E1 111.280} C_DIS
LIN {X -0.025,Y -610.645,Z 1229.417,A 0.000,B 0.000,C 90.000,E1 111.046} C_DIS
LIN {X 0.157,Y -614.609,Z 1229.412,A 0.000,B 0.000,C 90.000,E1 110.120} C_DIS
LIN {X 0.134,Y -615.311,Z 1229.411,A 0.000,B 0.000,C 90.000,E1 109.993} C_DIS
LIN {X 0.177,Y -618.477,Z 1229.407,A 0.000,B 0.000,C 90.000,E1 109.214} C_DIS
LIN {X -0.098,Y -620.297,Z 1229.404,A 0.000,B 0.000,C 90.000,E1 108.725} C_DIS
LIN {X 0.139,Y -626.498,Z 1229.396,A 0.000,B 0.000,C 90.000,E1 107.166} C_DIS
LIN {X 0.114,Y -627.479,Z 1229.394,A 0.000,B 0.000,C 90.000,E1 106.913} C_DIS
LIN {X -0.093,Y -628.664,Z 1229.393,A 0.000,B 0.000,C 90.000,E1 106.677} C_DIS
LIN {X 0.112,Y -630.639,Z 1229.390,A 0.000,B 0.000,C 90.000,E1 106.150} C_DIS
LIN {X 0.091,Y -631.800,Z 1229.388,A 0.000,B 0.000,C 90.000,E1 105.898} C_DIS
LIN {X 0.139,Y -634.578,Z 1229.384,A 0.000,B 0.000,C 90.000,E1 105.134} C_DIS
LIN {X -0.059,Y -636.220,Z 1229.381,A 0.000,B 0.000,C 90.000,E1 104.647} C_DIS
LIN {X 0.036,Y -638.056,Z 1229.377,A 0.000,B 0.000,C 90.000,E1 103.883} C_DIS
LIN {X 0.319,Y -639.086,Z 1229.374,A 0.000,B 0.000,C 90.000,E1 103.355} C_DIS
LIN {X -0.012,Y -639.806,Z 1229.372,A 0.000,B 0.000,C 90.000,E1 102.883} C_DIS
LIN {X 0.285,Y -640.219,Z 1229.369,A 0.000,B 0.000,C 90.000,E1 102.355} C_DIS
LIN {X 0.123,Y -640.340,Z 1229.367,A 0.000,B 0.000,C 90.000,E1 102.119} C_DIS
LIN {X -0.334,Y -640.148,Z 1229.365,A 0.000,B 0.000,C 90.000,E1 101.658} C_DIS
LIN {X -0.032,Y -639.695,Z 1229.362,A 0.000,B 0.000,C 90.000,E1 101.130} C_DIS
LIN {X -0.196,Y -639.347,Z 1229.360,A 0.000,B 0.000,C 90.000,E1 100.894} C_DIS
LIN {X 0.096,Y -638.274,Z 1229.358,A 0.000,B 0.000,C 90.000,E1 100.366} C_DIS
LIN {X 0.267,Y -636.885,Z 1229.355,A 0.000,B 0.000,C 90.000,E1 99.849} C_DIS
LIN {X -0.087,Y -635.050,Z 1229.352,A 0.000,B 0.000,C 90.000,E1 99.378} C_DIS
LIN {X 0.069,Y -632.797,Z 1229.349,A 0.000,B 0.000,C 90.000,E1 98.859} C_DIS
LIN {X 0.215,Y -630.350,Z 1229.346,A 0.000,B 0.000,C 90.000,E1 98.341} C_DIS
LIN {X -0.134,Y -628.190,Z 1229.344,A 0.000,B 0.000,C 90.000,E1 97.992} C_DIS
LIN {X 0.129,Y -625.777,Z 1229.342,A 0.000,B 0.000,C 90.000,E1 97.587} C_DIS
LIN {X 0.147,Y -620.850,Z 1229.339,A 0.000,B 0.000,C 90.000,E1 96.947} C_DIS
LIN {X -0.318,Y -617.488,Z 1229.337,A 0.000,B 0.000,C 90.000,E1 96.606} C_DIS
LIN {X -0.206,Y -611.186,Z 1229.333,A 0.000,B 0.000,C 90.000,E1 95.967} C_DIS
LIN {X 0.268,Y -604.232,Z 1229.330,A 0.000,B 0.000,C 90.000,E1 95.334} C_DIS
LIN {X -0.021,Y -596.433,Z 1229.327,A 0.000,B 0.000,C 90.000,E1 94.821} C_DIS
LIN {X 0.235,Y -588.578,Z 1229.324,A 0.000,B 0.000,C 90.000,E1 94.302} C_DIS
LIN {X -0.212,Y -583.578,Z 1229.323,A 0.000,B 0.000,C 90.000,E1 94.069} C_DIS
LIN {X -0.038,Y -576.735,Z 1229.321,A 0.000,B 0.000,C 90.000,E1 93.726} C_DIS
LIN {X -0.006,Y -571.555,Z 1229.319,A 0.000,B 0.000,C 90.000,E1 93.498} C_DIS
LIN {X 0.017,Y -566.579,Z 1229.318,A 0.000,B 0.000,C 90.000,E1 93.212} C_DIS
LIN {X -0.028,Y -566.553,Z 1229.318,A 0.000,B 0.000,C 90.000,E1 93.212} C_DIS
LIN {X -0.117,Y -565.458,Z 1229.317,A 0.000,B 0.000,C 90.000,E1 92.980} C_DIS
LIN {X -0.170,Y -565.450,Z 1229.317,A 0.000,B 0.000,C 90.000,E1 92.980} C_DIS
LIN {X -0.166,Y -565.180,Z 1229.314,A 0.000,B 0.000,C 90.000,E1 92.465} C_DIS
LIN {X -0.041,Y -565.537,Z 1229.308,A 0.000,B 0.000,C 90.000,E1 91.489} C_DIS
LIN {X 0.196,Y -566.882,Z 1229.298,A 0.000,B 0.000,C 90.000,E1 89.542} C_DIS
LIN {X -0.208,Y -568.041,Z 1229.288,A 0.000,B 0.000,C 90.000,E1 87.936} C_DIS
LIN {X 0.098,Y -569.523,Z 1229.278,A 0.000,B 0.000,C 90.000,E1 85.988} C_DIS
LIN {X 0.236,Y -571.722,Z 1229.264,A 0.000,B 0.000,C 90.000,E1 83.514} C_DIS
LIN {X 0.080,Y -573.281,Z 1229.255,A 0.000,B 0.000,C 90.000,E1 81.894} C_DIS
LIN {X -0.150,Y -574.488,Z 1229.248,A 0.000,B 0.000,C 90.000,E1 80.557} C_DIS
LIN {X 0.210,Y -575.483,Z 1229.240,A 0.000,B 0.000,C 90.000,E1 79.162} C_DIS
LIN {X -0.011,Y -576.725,Z 1229.229,A 0.000,B 0.000,C 90.000,E1 77.285} C_DIS
LIN {X 0.276,Y -577.371,Z 1229.223,A 0.000,B 0.000,C 90.000,E1 76.172} C_DIS
LIN {X 0.149,Y -578.007,Z 1229.217,A 0.000,B 0.000,C 90.000,E1 75.102} C_DIS
LIN {X -0.102,Y -578.882,Z 1229.208,A 0.000,B 0.000,C 90.000,E1 73.504} C_DIS
LIN {X 0.161,Y -579.625,Z 1229.201,A 0.000,B 0.000,C 90.000,E1 72.127} C_DIS
LIN {X -0.279,Y -580.623,Z 1229.192,A 0.000,B 0.000,C 90.000,E1 70.550} C_DIS
LIN {X -0.056,Y -582.128,Z 1229.178,A 0.000,B 0.000,C 90.000,E1 68.103} C_DIS
LIN {X -0.024,Y -583.474,Z 1229.169,A 0.000,B 0.000,C 90.000,E1 66.485} C_DIS
LIN {X -0.131,Y -584.693,Z 1229.162,A 0.000,B 0.000,C 90.000,E1 65.153} C_DIS
LIN {X -0.041,Y -586.610,Z 1229.150,A 0.000,B 0.000,C 90.000,E1 62.999} C_DIS
LIN {X 0.055,Y -588.259,Z 1229.141,A 0.000,B 0.000,C 90.000,E1 61.385} C_DIS
LIN {X -0.227,Y -589.635,Z 1229.134,A 0.000,B 0.000,C 90.000,E1 60.078} C_DIS
LIN {X -0.191,Y -591.011,Z 1229.126,A 0.000,B 0.000,C 90.000,E1 58.742} C_DIS
LIN {X 0.183,Y -592.256,Z 1229.119,A 0.000,B 0.000,C 90.000,E1 57.375} C_DIS
LIN {X -0.238,Y -593.439,Z 1229.112,A 0.000,B 0.000,C 90.000,E1 56.087} C_DIS
LIN {X -0.316,Y -594.520,Z 1229.104,A 0.000,B 0.000,C 90.000,E1 54.769} C_DIS
LIN {X -0.030,Y -595.579,Z 1229.097,A 0.000,B 0.000,C 90.000,E1 53.417} C_DIS
LIN {X 0.263,Y -597.003,Z 1229.087,A 0.000,B 0.000,C 90.000,E1 51.537} C_DIS
LIN {X -0.349,Y -597.591,Z 1229.082,A 0.000,B 0.000,C 90.000,E1 50.803} C_DIS
LIN {X 0.123,Y -598.522,Z 1229.070,A 0.000,B 0.000,C 90.000,E1 48.647} C_DIS
LIN {X -0.308,Y -599.021,Z 1229.065,A 0.000,B 0.000,C 90.000,E1 47.634} C_DIS
LIN {X -0.098,Y -599.327,Z 1229.057,A 0.000,B 0.000,C 90.000,E1 46.296} C_DIS
LIN {X -0.101,Y -599.401,Z 1229.051,A 0.000,B 0.000,C 90.000,E1 45.243} C_DIS
LIN {X -0.101,Y -599.297,Z 1229.046,A 0.000,B 0.000,C 90.000,E1 44.190} C_DIS
LIN {X -0.108,Y -599.031,Z 1229.040,A 0.000,B 0.000,C 90.000,E1 43.137} C_DIS
LIN {X 0.127,Y -598.700,Z 1229.035,A 0.000,B 0.000,C 90.000,E1 42.324} C_DIS
LIN {X 0.103,Y -597.837,Z 1229.026,A 0.000,B 0.000,C 90.000,E1 40.744} C_DIS
LIN {X -0.043,Y -597.164,Z 1229.019,A 0.000,B 0.000,C 90.000,E1 39.439} C_DIS
LIN {X -0.047,Y -596.320,Z 1229.013,A 0.000,B 0.000,C 90.000,E1 38.382} C_DIS
LIN {X -0.213,Y -594.923,Z 1229.006,A 0.000,B 0.000,C 90.000,E1 37.076} C_DIS
LIN {X -0.150,Y -593.588,Z 1229.000,A 0.000,B 0.000,C 90.000,E1 36.011} C_DIS
LIN {X 0.162,Y -592.341,Z 1228.996,A 0.000,B 0.000,C 90.000,E1 35.185} C_DIS
LIN {X -0.022,Y -590.914,Z 1228.991,A 0.000,B 0.000,C 90.000,E1 34.405} C_DIS
LIN {X -0.351,Y -588.679,Z 1228.985,A 0.000,B 0.000,C 90.000,E1 33.372} C_DIS
LIN {X 0.097,Y -585.956,Z 1228.979,A 0.000,B 0.000,C 90.000,E1 32.260} C_DIS
LIN {X -0.161,Y -584.341,Z 1228.976,A 0.000,B 0.000,C 90.000,E1 31.750} C_DIS
LIN {X 0.048,Y -581.650,Z 1228.972,A 0.000,B 0.000,C 90.000,E1 30.924} C_DIS
LIN {X -0.075,Y -578.515,Z 1228.967,A 0.000,B 0.000,C 90.000,E1 30.129} C_DIS
LIN {X -0.154,Y -575.591,Z 1228.964,A 0.000,B 0.000,C 90.000,E1 29.461} C_DIS
LIN {X 0.040,Y -572.992,Z 1228.961,A 0.000,B 0.000,C 90.000,E1 28.899} C_DIS
LIN {X -0.009,Y -570.199,Z 1228.958,A 0.000,B 0.000,C 90.000,E1 28.359} C_DIS
LIN {X 0.149,Y -564.901,Z 1228.952,A 0.000,B 0.000,C 90.000,E1 27.385} C_DIS
LIN {X -0.320,Y -560.644,Z 1228.948,A 0.000,B 0.000,C 90.000,E1 26.744} C_DIS
LIN {X 0.029,Y -557.010,Z 1228.945,A 0.000,B 0.000,C 90.000,E1 26.155} C_DIS
LIN {X 0.118,Y -553.218,Z 1228.942,A 0.000,B 0.000,C 90.000,E1 25.591} C_DIS
LIN {X -0.214,Y -550.206,Z 1228.940,A 0.000,B 0.000,C 90.000,E1 25.207} C_DIS
LIN {X 0.067,Y -543.458,Z 1228.935,A 0.000,B 0.000,C 90.000,E1 24.335} C_DIS
LIN {X -0.084,Y -537.501,Z 1228.931,A 0.000,B 0.000,C 90.000,E1 23.643} C_DIS
LIN {X 0.204,Y -531.196,Z 1228.927,A 0.000,B 0.000,C 90.000,E1 22.898} C_DIS
LIN {X -0.024,Y -522.171,Z 1228.922,A 0.000,B 0.000,C 90.000,E1 21.950} C_DIS
LIN {X 0.088,Y -512.771,Z 1228.917,A 0.000,B 0.000,C 90.000,E1 20.972} C_DIS
LIN {X -0.057,Y -507.140,Z 1228.913,A 0.000,B 0.000,C 90.000,E1 20.429} C_DIS
LIN {X -0.132,Y -498.802,Z 1228.909,A 0.000,B 0.000,C 90.000,E1 19.631} C_DIS
LIN {X 0.223,Y -490.177,Z 1228.905,A 0.000,B 0.000,C 90.000,E1 18.779} C_DIS
LIN {X -0.137,Y -481.653,Z 1228.900,A 0.000,B 0.000,C 90.000,E1 18.055} C_DIS
LIN {X -0.011,Y -469.697,Z 1228.894,A 0.000,B 0.000,C 90.000,E1 16.985} C_DIS
LIN {X -0.148,Y -453.578,Z 1228.886,A 0.000,B 0.000,C 90.000,E1 15.552} C_DIS
LIN {X 0.107,Y -430.448,Z 1228.874,A 0.000,B 0.000,C 90.000,E1 13.300} C_DIS
LIN {X 0.063,Y -413.328,Z 1228.864,A 0.000,B 0.000,C 90.000,E1 11.478} C_DIS
LIN {X 0.138,Y -402.319,Z 1228.857,A 0.000,B 0.000,C 90.000,E1 10.197} C_DIS
LIN {X -0.092,Y -398.493,Z 1228.854,A 0.000,B 0.000,C 90.000,E1 9.726} C_DIS
LIN {X -0.069,Y -395.188,Z 1228.851,A 0.000,B 0.000,C 90.000,E1 9.208} C_DIS
LIN {X 0.054,Y -394.030,Z 1228.849,A 0.000,B 0.000,C 90.000,E1 8.859} C_DIS
LIN {X 0.016,Y -394.027,Z 1228.849,A 0.000,B 0.000,C 90.000,E1 8.859} C_DIS
LIN {X -0.048,Y -394.070,Z 1228.848,A 0.000,B 0.000,C 90.000,E1 8.681} C_DIS
LIN {X -0.085,Y -394.092,Z 1228.848,A 0.000,B 0.000,C 90.000,E1 8.681} C_DIS
LIN {X 0.002,Y -396.869,Z 1228.845,A 0.000,B 0.000,C 90.000,E1 8.049} C_DIS
LIN {X 0.065,Y -400.336,Z 1228.843,A 0.000,B 0.000,C 90.000,E1 7.644} C_DIS
LIN {X -0.043,Y -404.079,Z 1228.841,A 0.000,B 0.000,C 90.000,E1 7.352} C_DIS
LIN {X 0.118,Y -419.863,Z 1228.834,A 0.000,B 0.000,C 90.000,E1 6.144} C_DIS
LIN {X -0.107,Y -425.759,Z 1228.832,A 0.000,B 0.000,C 90.000,E1 5.739} C_DIS
LIN {X -0.022,Y -436.874,Z 1228.827,A 0.000,B 0.000,C 90.000,E1 4.878} C_DIS
LIN {X -0.068,Y -451.061,Z 1228.821,A 0.000,B 0.000,C 90.000,E1 3.784} C_DIS
LIN {X 0.093,Y -460.423,Z 1228.817,A 0.000,B 0.000,C 90.000,E1 3.037} C_DIS
LIN {X 0.209,Y -468.119,Z 1228.814,A 0.000,B 0.000,C 90.000,E1 2.407} C_DIS
LIN {X -0.041,Y -472.605,Z 1228.812,A 0.000,B 0.000,C 90.000,E1 2.064} C_DIS
LIN {X -0.073,Y -478.445,Z 1228.809,A 0.000,B 0.000,C 90.000,E1 1.547} C_DIS
LIN {X 0.050,Y -485.408,Z 1228.805,A 0.000,B 0.000,C 90.000,E1 0.859} C_DIS
LIN {X 0.109,Y -491.929,Z 1228.801,A 0.000,B 0.000,C 90.000,E1 0.172} C_DIS
LIN {X 0.148,Y -498.080,Z 1228.797,A 0.000,B 0.000,C 90.000,E1 359.484} C_DIS
LIN {X 0.098,Y -504.232,Z 1228.793,A 0.000,B 0.000,C 90.000,E1 358.740} C_DIS
LIN {X 0.096,Y -509.900,Z 1228.789,A 0.000,B 0.000,C 90.000,E1 357.993} C_DIS
LIN {X 0.133,Y -515.073,Z 1228.785,A 0.000,B 0.000,C 90.000,E1 357.249} C_DIS
LIN {X 0.013,Y -518.993,Z 1228.782,A 0.000,B 0.000,C 90.000,E1 356.674} C_DIS
LIN {X 0.158,Y -523.525,Z 1228.777,A 0.000,B 0.000,C 90.000,E1 355.927} C_DIS
LIN {X -0.219,Y -527.600,Z 1228.773,A 0.000,B 0.000,C 90.000,E1 355.241} C_DIS
LIN {X 0.052,Y -531.333,Z 1228.769,A 0.000,B 0.000,C 90.000,E1 354.489} C_DIS
LIN {X 0.056,Y -534.115,Z 1228.766,A 0.000,B 0.000,C 90.000,E1 353.913} C_DIS
LIN {X 0.081,Y -536.662,Z 1228.763,A 0.000,B 0.000,C 90.000,E1 353.337} C_DIS
LIN {X 0.182,Y -540.151,Z 1228.758,A 0.000,B 0.000,C 90.000,E1 352.470} C_DIS
LIN {X 0.243,Y -542.334,Z 1228.755,A 0.000,B 0.000,C 90.000,E1 351.894} C_DIS
LIN {X -0.139,Y -545.263,Z 1228.750,A 0.000,B 0.000,C 90.000,E1 351.084} C_DIS
LIN {X 0.137,Y -548.005,Z 1228.746,A 0.000,B 0.000,C 90.000,E1 350.208} C_DIS
LIN {X -0.192,Y -550.380,Z 1228.741,A 0.000,B 0.000,C 90.000,E1 349.398} C_DIS
LIN {X -0.159,Y -554.049,Z 1228.733,A 0.000,B 0.000,C 90.000,E1 347.993} C_DIS
LIN {X 0.218,Y -556.095,Z 1228.729,A 0.000,B 0.000,C 90.000,E1 347.117} C_DIS
LIN {X -0.064,Y -559.084,Z 1228.721,A 0.000,B 0.000,C 90.000,E1 345.755} C_DIS
LIN {X -0.186,Y -560.753,Z 1228.716,A 0.000,B 0.000,C 90.000,E1 344.936} C_DIS
LIN {X 0.154,Y -562.773,Z 1228.710,A 0.000,B 0.000,C 90.000,E1 343.795} C_DIS
LIN {X 0.144,Y -564.964,Z 1228.702,A 0.000,B 0.000,C 90.000,E1 342.417} C_DIS
LIN {X 0.225,Y -566.090,Z 1228.698,A 0.000,B 0.000,C 90.000,E1 341.583} C_DIS
LIN {X -0.040,Y -567.153,Z 1228.693,A 0.000,B 0.000,C 90.000,E1 340.786} C_DIS
LIN {X 0.247,Y -567.957,Z 1228.689,A 0.000,B 0.000,C 90.000,E1 339.934} C_DIS
LIN {X 0.008,Y -568.550,Z 1228.684,A 0.000,B 0.000,C 90.000,E1 339.135} C_DIS
LIN {X 0.306,Y -568.901,Z 1228.680,A 0.000,B 0.000,C 90.000,E1 338.284} C_DIS
LIN {X 0.073,Y -568.992,Z 1228.675,A 0.000,B 0.000,C 90.000,E1 337.486} C_DIS
LIN {X -0.117,Y -568.500,Z 1228.669,A 0.000,B 0.000,C 90.000,E1 336.410} C_DIS
LIN {X -0.361,Y -567.752,Z 1228.664,A 0.000,B 0.000,C 90.000,E1 335.613} C_DIS
LIN {X -0.204,Y -567.124,Z 1228.661,A 0.000,B 0.000,C 90.000,E1 335.049} C_DIS
LIN {X 0.010,Y -565.779,Z 1228.657,A 0.000,B 0.000,C 90.000,E1 334.204} C_DIS
LIN {X 0.153,Y -564.748,Z 1228.654,A 0.000,B 0.000,C 90.000,E1 333.640} C_DIS
LIN {X 0.093,Y -562.789,Z 1228.649,A 0.000,B 0.000,C 90.000,E1 332.820} C_DIS
LIN {X -0.229,Y -560.600,Z 1228.645,A 0.000,B 0.000,C 90.000,E1 332.025} C_DIS
LIN {X 0.130,Y -558.789,Z 1228.641,A 0.000,B 0.000,C 90.000,E1 331.435} C_DIS
LIN {X -0.281,Y -556.621,Z 1228.638,A 0.000,B 0.000,C 90.000,E1 330.923} C_DIS
LIN {X -0.064,Y -553.565,Z 1228.635,A 0.000,B 0.000,C 90.000,E1 330.205} C_DIS
LIN {X 0.118,Y -550.075,Z 1228.631,A 0.000,B 0.000,C 90.000,E1 329.488} C_DIS
LIN {X -0.084,Y -546.803,Z 1228.627,A 0.000,B 0.000,C 90.000,E1 328.948} C_DIS
LIN {X -0.178,Y -544.187,Z 1228.625,A 0.000,B 0.000,C 90.000,E1 328.535} C_DIS
LIN {X 0.197,Y -539.479,Z 1228.621,A 0.000,B 0.000,C 90.000,E1 327.788} C_DIS
LIN {X -0.217,Y -534.396,Z 1228.617,A 0.000,B 0.000,C 90.000,E1 327.120} C_DIS
LIN {X 0.197,Y -527.774,Z 1228.612,A 0.000,B 0.000,C 90.000,E1 326.215} C_DIS
LIN {X -0.072,Y -516.737,Z 1228.604,A 0.000,B 0.000,C 90.000,E1 324.815} C_DIS
LIN {X 0.048,Y -513.259,Z 1228.602,A 0.000,B 0.000,C 90.000,E1 324.276} C_DIS
LIN {X 0.005,Y -510.786,Z 1228.599,A 0.000,B 0.000,C 90.000,E1 323.783} C_DIS
LIN {X 0.025,Y -509.629,Z 1228.597,A 0.000,B 0.000,C 90.000,E1 323.463} C_DIS
LIN {X -0.061,Y -508.680,Z 1228.595,A 0.000,B 0.000,C 90.000,E1 323.176} C_DIS
LIN {X 0.257,Y -508.124,Z 1228.594,A 0.000,B 0.000,C 90.000,E1 322.844} C_DIS
LIN {X 0.068,Y -507.233,Z 1228.590,A 0.000,B 0.000,C 90.000,E1 322.271} C_DIS
LIN {X 0.088,Y -506.649,Z 1228.586,A 0.000,B 0.000,C 90.000,E1 321.376} C_DIS
LIN {X -0.099,Y -506.989,Z 1228.577,A 0.000,B 0.000,C 90.000,E1 319.908} C_DIS
LIN {X 0.276,Y -508.031,Z 1228.567,A 0.000,B 0.000,C 90.000,E1 318.081} C_DIS
LIN {X 0.162,Y -508.705,Z 1228.561,A 0.000,B 0.000,C 90.000,E1 316.905} C_DIS
LIN {X -0.056,Y -509.354,Z 1228.552,A 0.000,B 0.000,C 90.000,E1 315.445} C_DIS
LIN {X 0.085,Y -509.911,Z 1228.544,A 0.000,B 0.000,C 90.000,E1 313.947} C_DIS
LIN {X 0.010,Y -510.789,Z 1228.533,A 0.000,B 0.000,C 90.000,E1 311.881} C_DIS
LIN {X -0.025,Y -511.296,Z 1228.526,A 0.000,B 0.000,C 90.000,E1 310.701} C_DIS
LIN {X 0.199,Y -511.839,Z 1228.518,A 0.000,B 0.000,C 90.000,E1 309.197} C_DIS
LIN {X 0.025,Y -512.409,Z 1228.508,A 0.000,B 0.000,C 90.000,E1 307.443} C_DIS
LIN {X -0.035,Y -512.936,Z 1228.498,A 0.000,B 0.000,C 90.000,E1 305.678} C_DIS
LIN {X -0.085,Y -513.483,Z 1228.488,A 0.000,B 0.000,C 90.000,E1 303.913} C_DIS
LIN {X 0.007,Y -513.921,Z 1228.479,A 0.000,B 0.000,C 90.000,E1 302.133} C_DIS
LIN {X -0.170,Y -514.105,Z 1228.469,A 0.000,B 0.000,C 90.000,E1 300.384} C_DIS
LIN {X 0.188,Y -514.245,Z 1228.461,A 0.000,B 0.000,C 90.000,E1 298.871} C_DIS
LIN {X -0.040,Y -514.338,Z 1228.451,A 0.000,B 0.000,C 90.000,E1 297.129} C_DIS
LIN {X -0.031,Y -514.425,Z 1228.438,A 0.000,B 0.000,C 90.000,E1 294.771} C_DIS
LIN {X -0.005,Y -514.532,Z 1228.431,A 0.000,B 0.000,C 90.000,E1 293.590} C_DIS
LIN {X 0.157,Y -514.456,Z 1228.423,A 0.000,B 0.000,C 90.000,E1 292.099} C_DIS
LIN {X 0.059,Y -514.138,Z 1228.418,A 0.000,B 0.000,C 90.000,E1 291.227} C_DIS
LIN {X -0.106,Y -513.722,Z 1228.411,A 0.000,B 0.000,C 90.000,E1 290.066} C_DIS
LIN {X -0.091,Y -512.765,Z 1228.400,A 0.000,B 0.000,C 90.000,E1 288.000} C_DIS
LIN {X 0.154,Y -512.095,Z 1228.392,A 0.000,B 0.000,C 90.000,E1 286.496} C_DIS
LIN {X 0.238,Y -511.404,Z 1228.384,A 0.000,B 0.000,C 90.000,E1 285.009} C_DIS
LIN {X 0.223,Y -510.148,Z 1228.372,A 0.000,B 0.000,C 90.000,E1 282.939} C_DIS
LIN {X -0.051,Y -508.709,Z 1228.361,A 0.000,B 0.000,C 90.000,E1 280.894} C_DIS
LIN {X 0.053,Y -507.244,Z 1228.349,A 0.000,B 0.000,C 90.000,E1 278.803} C_DIS
LIN {X -0.136,Y -505.568,Z 1228.334,A 0.000,B 0.000,C 90.000,E1 276.144} C_DIS
LIN {X 0.131,Y -504.227,Z 1228.321,A 0.000,B 0.000,C 90.000,E1 273.726} C_DIS
LIN {X 0.099,Y -503.313,Z 1228.313,A 0.000,B 0.000,C 90.000,E1 272.236} C_DIS
LIN {X 0.165,Y -502.456,Z 1228.306,A 0.000,B 0.000,C 90.000,E1 271.031} C_DIS
LIN {X -0.147,Y -501.082,Z 1228.294,A 0.000,B 0.000,C 90.000,E1 268.969} C_DIS
LIN {X 0.139,Y -500.032,Z 1228.284,A 0.000,B 0.000,C 90.000,E1 267.135} C_DIS
LIN {X 0.152,Y -499.357,Z 1228.278,A 0.000,B 0.000,C 90.000,E1 265.931} C_DIS
LIN {X 0.191,Y -498.603,Z 1228.271,A 0.000,B 0.000,C 90.000,E1 264.723} C_DIS
LIN {X 0.220,Y -497.756,Z 1228.264,A 0.000,B 0.000,C 90.000,E1 263.514} C_DIS
LIN {X 0.205,Y -496.402,Z 1228.256,A 0.000,B 0.000,C 90.000,E1 262.008} C_DIS
LIN {X 0.082,Y -494.737,Z 1228.246,A 0.000,B 0.000,C 90.000,E1 260.208} C_DIS
LIN {X -0.181,Y -492.651,Z 1228.232,A 0.000,B 0.000,C 90.000,E1 257.813} C_DIS
LIN {X 0.063,Y -490.958,Z 1228.219,A 0.000,B 0.000,C 90.000,E1 255.353} C_DIS
LIN {X 0.141,Y -489.452,Z 1228.205,A 0.000,B 0.000,C 90.000,E1 252.906} C_DIS
LIN {X -0.028,Y -488.553,Z 1228.195,A 0.000,B 0.000,C 90.000,E1 251.094} C_DIS
LIN {X -0.075,Y -487.813,Z 1228.187,A 0.000,B 0.000,C 90.000,E1 249.571} C_DIS
LIN {X 0.037,Y -486.987,Z 1228.178,A 0.000,B 0.000,C 90.000,E1 248.028} C_DIS
LIN {X 0.132,Y -485.980,Z 1228.170,A 0.000,B 0.000,C 90.000,E1 246.485} C_DIS
LIN {X -0.050,Y -484.763,Z 1228.161,A 0.000,B 0.000,C 90.000,E1 244.973} C_DIS
LIN {X 0.164,Y -482.672,Z 1228.147,A 0.000,B 0.000,C 90.000,E1 242.487} C_DIS
LIN {X -0.070,Y -481.207,Z 1228.139,A 0.000,B 0.000,C 90.000,E1 240.973} C_DIS
LIN {X -0.120,Y -479.869,Z 1228.132,A 0.000,B 0.000,C 90.000,E1 239.744} C_DIS
LIN {X 0.033,Y -477.837,Z 1228.122,A 0.000,B 0.000,C 90.000,E1 237.867} C_DIS
LIN {X 0.219,Y -476.839,Z 1228.116,A 0.000,B 0.000,C 90.000,E1 236.914} C_DIS
LIN {X 0.155,Y -474.788,Z 1228.106,A 0.000,B 0.000,C 90.000,E1 235.055} C_DIS
LIN {X 0.143,Y -473.140,Z 1228.097,A 0.000,B 0.000,C 90.000,E1 233.497} C_DIS
LIN {X -0.057,Y -470.974,Z 1228.085,A 0.000,B 0.000,C 90.000,E1 231.331} C_DIS
LIN {X 0.039,Y -468.799,Z 1228.071,A 0.000,B 0.000,C 90.000,E1 228.809} C_DIS
LIN {X 0.162,Y -467.173,Z 1228.061,A 0.000,B 0.000,C 90.000,E1 226.905} C_DIS
LIN {X -0.145,Y -463.999,Z 1228.026,A 0.000,B 0.000,C 90.000,E1 220.620} C_DIS
LIN {X 0.140,Y -465.262,Z 1227.997,A 0.000,B 0.000,C 90.000,E1 215.518} C_DIS
LIN {X -0.044,Y -467.779,Z 1227.976,A 0.000,B 0.000,C 90.000,E1 211.750} C_DIS
LIN {X -0.063,Y -469.310,Z 1227.968,A 0.000,B 0.000,C 90.000,E1 210.178} C_DIS
LIN {X 0.097,Y -472.452,Z 1227.952,A 0.000,B 0.000,C 90.000,E1 207.334} C_DIS
LIN {X 0.026,Y -475.177,Z 1227.940,A 0.000,B 0.000,C 90.000,E1 205.155} C_DIS
LIN {X 0.198,Y -480.351,Z 1227.921,A 0.000,B 0.000,C 90.000,E1 201.716} C_DIS
LIN {X 0.022,Y -484.864,Z 1227.907,A 0.000,B 0.000,C 90.000,E1 199.268} C_DIS
LIN {X 0.259,Y -489.451,Z 1227.895,A 0.000,B 0.000,C 90.000,E1 197.094} C_DIS
LIN {X -0.241,Y -495.230,Z 1227.882,A 0.000,B 0.000,C 90.000,E1 194.717} C_DIS
LIN {X 0.026,Y -499.162,Z 1227.873,A 0.000,B 0.000,C 90.000,E1 193.175} C_DIS
LIN {X 0.145,Y -503.157,Z 1227.865,A 0.000,B 0.000,C 90.000,E1 191.658} C_DIS
LIN {X 0.208,Y -509.784,Z 1227.852,A 0.000,B 0.000,C 90.000,E1 189.265} C_DIS
LIN {X -0.027,Y -513.229,Z 1227.845,A 0.000,B 0.000,C 90.000,E1 188.106} C_DIS
LIN {X 0.188,Y -518.240,Z 1227.835,A 0.000,B 0.000,C 90.000,E1 186.315} C_DIS
LIN {X -0.051,Y -522.394,Z 1227.827,A 0.000,B 0.000,C 90.000,E1 184.878} C_DIS
LIN {X -0.212,Y -526.532,Z 1227.819,A 0.000,B 0.000,C 90.000,E1 183.440} C_DIS
LIN {X 0.199,Y -530.694,Z 1227.811,A 0.000,B 0.000,C 90.000,E1 181.949} C_DIS
LIN {X 0.155,Y -534.719,Z 1227.803,A 0.000,B 0.000,C 90.000,E1 180.516} C_DIS
LIN {X 0.172,Y -538.742,Z 1227.795,A 0.000,B 0.000,C 90.000,E1 179.083} C_DIS
LIN {X 0.273,Y -542.613,Z 1227.787,A 0.000,B 0.000,C 90.000,E1 177.650} C_DIS
LIN {X -0.163,Y -544.880,Z 1227.782,A 0.000,B 0.000,C 90.000,E1 176.846} C_DIS
LIN {X 0.128,Y -549.191,Z 1227.773,A 0.000,B 0.000,C 90.000,E1 175.122} C_DIS
LIN {X -0.095,Y -552.677,Z 1227.765,A 0.000,B 0.000,C 90.000,E1 173.742} C_DIS
LIN {X -0.078,Y -556.658,Z 1227.756,A 0.000,B 0.000,C 90.000,E1 172.064} C_DIS
LIN {X -0.259,Y -559.275,Z 1227.750,A 0.000,B 0.000,C 90.000,E1 170.971} C_DIS
LIN {X -0.075,Y -562.540,Z 1227.742,A 0.000,B 0.000,C 90.000,E1 169.567} C_DIS
LIN {X 0.069,Y -565.725,Z 1227.734,A 0.000,B 0.000,C 90.000,E1 168.173} C_DIS
LIN {X 0.312,Y -570.253,Z 1227.724,A 0.000,B 0.000,C 90.000,E1 166.228} C_DIS
LIN {X 0.116,Y -574.979,Z 1227.713,A 0.000,B 0.000,C 90.000,E1 164.338} C_DIS
LIN {X 0.025,Y -586.852,Z 1227.691,A 0.000,B 0.000,C 90.000,E1 160.296} C_DIS
LIN {X 0.033,Y -598.959,Z 1227.673,A 0.000,B 0.000,C 90.000,E1 157.102} C_DIS
LIN {X -0.160,Y -606.337,Z 1227.663,A 0.000,B 0.000,C 90.000,E1 155.281} C_DIS
LIN {X -0.115,Y -611.463,Z 1227.655,A 0.000,B 0.000,C 90.000,E1 153.973} C_DIS
LIN {X 0.003,Y -616.399,Z 1227.648,A 0.000,B 0.000,C 90.000,E1 152.666} C_DIS
LIN {X -0.083,Y -621.911,Z 1227.640,A 0.000,B 0.000,C 90.000,E1 151.129} C_DIS
LIN {X 0.213,Y -624.682,Z 1227.635,A 0.000,B 0.000,C 90.000,E1 150.333} C_DIS
LIN {X 0.023,Y -629.179,Z 1227.628,A 0.000,B 0.000,C 90.000,E1 149.076} C_DIS
LIN {X -0.279,Y -634.423,Z 1227.620,A 0.000,B 0.000,C 90.000,E1 147.582} C_DIS
LIN {X 0.407,Y -639.271,Z 1227.611,A 0.000,B 0.000,C 90.000,E1 146.008} C_DIS
LIN {X -0.153,Y -642.263,Z 1227.606,A 0.000,B 0.000,C 90.000,E1 145.055} C_DIS
LIN {X 0.065,Y -645.102,Z 1227.600,A 0.000,B 0.000,C 90.000,E1 144.036} C_DIS
LIN {X 0.042,Y -647.054,Z 1227.596,A 0.000,B 0.000,C 90.000,E1 143.290} C_DIS
LIN {X -0.145,Y -650.052,Z 1227.589,A 0.000,B 0.000,C 90.000,E1 142.065} C_DIS
LIN {X -0.406,Y -654.122,Z 1227.580,A 0.000,B 0.000,C 90.000,E1 140.356} C_DIS
LIN {X -0.025,Y -656.290,Z 1227.574,A 0.000,B 0.000,C 90.000,E1 139.337} C_DIS
LIN {X -0.216,Y -660.186,Z 1227.565,A 0.000,B 0.000,C 90.000,E1 137.634} C_DIS
LIN {X 0.123,Y -665.155,Z 1227.552,A 0.000,B 0.000,C 90.000,E1 135.405} C_DIS
LIN {X 0.116,Y -668.188,Z 1227.546,A 0.000,B 0.000,C 90.000,E1 134.190} C_DIS
LIN {X 0.248,Y -673.743,Z 1227.533,A 0.000,B 0.000,C 90.000,E1 132.000} C_DIS
LIN {X -0.098,Y -676.729,Z 1227.527,A 0.000,B 0.000,C 90.000,E1 130.825} C_DIS
LIN {X -0.329,Y -679.786,Z 1227.520,A 0.000,B 0.000,C 90.000,E1 129.644} C_DIS
LIN {X 0.061,Y -683.434,Z 1227.512,A 0.000,B 0.000,C 90.000,E1 128.177} C_DIS
LIN {X 0.106,Y -687.026,Z 1227.504,A 0.000,B 0.000,C 90.000,E1 126.744} C_DIS
LIN {X -0.011,Y -689.308,Z 1227.499,A 0.000,B 0.000,C 90.000,E1 125.804} C_DIS
LIN {X -0.263,Y -692.545,Z 1227.491,A 0.000,B 0.000,C 90.000,E1 124.405} C_DIS
LIN {X -0.142,Y -694.662,Z 1227.486,A 0.000,B 0.000,C 90.000,E1 123.452} C_DIS
LIN {X 0.038,Y -697.218,Z 1227.479,A 0.000,B 0.000,C 90.000,E1 122.260} C_DIS
LIN {X -0.152,Y -699.050,Z 1227.474,A 0.000,B 0.000,C 90.000,E1 121.337} C_DIS
LIN {X 0.045,Y -700.879,Z 1227.469,A 0.000,B 0.000,C 90.000,E1 120.384} C_DIS
LIN {X 0.179,Y -702.986,Z 1227.462,A 0.000,B 0.000,C 90.000,E1 119.205} C_DIS
LIN {X 0.064,Y -704.418,Z 1227.457,A 0.000,B 0.000,C 90.000,E1 118.281} C_DIS
LIN {X -0.318,Y -704.999,Z 1227.455,A 0.000,B 0.000,C 90.000,E1 117.847} C_DIS
LIN {X -0.077,Y -705.643,Z 1227.451,A 0.000,B 0.000,C 90.000,E1 117.129} C_DIS
LIN {X 0.145,Y -706.219,Z 1227.446,A 0.000,B 0.000,C 90.000,E1 116.181} C_DIS
LIN {X 0.098,Y -706.352,Z 1227.443,A 0.000,B 0.000,C 90.000,E1 115.720} C_DIS
LIN {X 0.037,Y -706.162,Z 1227.439,A 0.000,B 0.000,C 90.000,E1 115.027} C_DIS
LIN {X -0.315,Y -705.882,Z 1227.437,A 0.000,B 0.000,C 90.000,E1 114.591} C_DIS
LIN {X 0.266,Y -705.027,Z 1227.434,A 0.000,B 0.000,C 90.000,E1 114.079} C_DIS
LIN {X -0.377,Y -704.442,Z 1227.433,A 0.000,B 0.000,C 90.000,E1 113.898} C_DIS
LIN {X 0.191,Y -702.331,Z 1227.430,A 0.000,B 0.000,C 90.000,E1 113.387} C_DIS
LIN {X 0.329,Y -701.709,Z 1227.429,A 0.000,B 0.000,C 90.000,E1 113.259} C_DIS
LIN {X 0.191,Y -700.768,Z 1227.429,A 0.000,B 0.000,C 90.000,E1 113.153} C_DIS
LIN {X 0.019,Y -695.585,Z 1227.426,A 0.000,B 0.000,C 90.000,E1 112.717} C_DIS
LIN {X 0.236,Y -693.935,Z 1227.426,A 0.000,B 0.000,C 90.000,E1 112.589} C_DIS
LIN {X -0.188,Y -691.040,Z 1227.425,A 0.000,B 0.000,C 90.000,E1 112.514} C_DIS
LIN {X 0.200,Y -686.446,Z 1227.424,A 0.000,B 0.000,C 90.000,E1 112.333} C_DIS
LIN {X -0.230,Y -684.478,Z 1227.424,A 0.000,B 0.000,C 90.000,E1 112.333} C_DIS
LIN {X -0.075,Y -676.654,Z 1227.424,A 0.000,B 0.000,C 90.000,E1 112.280} C_DIS
LIN {X -0.108,Y -616.008,Z 1227.424,A 0.000,B 0.000,C 90.000,E1 112.280} C_DIS
LIN {X 0.139,Y -612.671,Z 1227.423,A 0.000,B 0.000,C 90.000,E1 112.078} C_DIS
LIN {X -0.061,Y -610.251,Z 1227.422,A 0.000,B 0.000,C 90.000,E1 111.897} C_DIS
LIN {X -0.085,Y -609.732,Z 1227.421,A 0.000,B 0.000,C 90.000,E1 111.844} C_DIS
LIN {X -0.162,Y -608.046,Z 1227.420,A 0.000,B 0.000,C 90.000,E1 111.589} C_DIS
LIN {X -0.206,Y -608.031,Z 1227.420,A 0.000,B 0.000,C 90.000,E1 111.589} C_DIS
LIN {X -0.214,Y -608.234,Z 1227.418,A 0.000,B 0.000,C 90.000,E1 111.280} C_DIS
LIN {X -0.215,Y -610.744,Z 1227.414,A 0.000,B 0.000,C 90.000,E1 110.610} C_DIS
LIN {X -0.012,Y -614.169,Z 1227.410,A 0.000,B 0.000,C 90.000,E1 109.812} C_DIS
LIN {X 0.266,Y -616.275,Z 1227.407,A 0.000,B 0.000,C 90.000,E1 109.268} C_DIS
LIN {X 0.303,Y -627.215,Z 1227.392,A 0.000,B 0.000,C 90.000,E1 106.441} C_DIS
LIN {X -0.131,Y -630.184,Z 1227.387,A 0.000,B 0.000,C 90.000,E1 105.717} C_DIS
LIN {X 0.089,Y -632.040,Z 1227.385,A 0.000,B 0.000,C 90.000,E1 105.190} C_DIS
LIN {X -0.286,Y -633.572,Z 1227.382,A 0.000,B 0.000,C 90.000,E1 104.717} C_DIS
LIN {X -0.061,Y -635.435,Z 1227.377,A 0.000,B 0.000,C 90.000,E1 103.939} C_DIS
LIN {X 0.202,Y -636.388,Z 1227.375,A 0.000,B 0.000,C 90.000,E1 103.411} C_DIS
LIN {X -0.146,Y -637.151,Z 1227.372,A 0.000,B 0.000,C 90.000,E1 102.939} C_DIS
LIN {X 0.302,Y -637.412,Z 1227.370,A 0.000,B 0.000,C 90.000,E1 102.647} C_DIS
LIN {X -0.042,Y -637.622,Z 1227.368,A 0.000,B 0.000,C 90.000,E1 102.175} C_DIS
LIN {X 0.109,Y -637.366,Z 1227.365,A 0.000,B 0.000,C 90.000,E1 101.658} C_DIS
LIN {X -0.234,Y -636.852,Z 1227.362,A 0.000,B 0.000,C 90.000,E1 101.186} C_DIS
LIN {X 0.218,Y -636.443,Z 1227.361,A 0.000,B 0.000,C 90.000,E1 100.894} C_DIS
LIN {X -0.136,Y -635.359,Z 1227.358,A 0.000,B 0.000,C 90.000,E1 100.423} C_DIS
LIN {X 0.015,Y -633.988,Z 1227.355,A 0.000,B 0.000,C 90.000,E1 99.905} C_DIS
LIN {X 0.266,Y -632.209,Z 1227.352,A 0.000,B 0.000,C 90.000,E1 99.378} C_DIS
LIN {X 0.202,Y -628.838,Z 1227.348,A 0.000,B 0.000,C 90.000,E1 98.624} C_DIS
LIN {X -0.155,Y -626.838,Z 1227.346,A 0.000,B 0.000,C 90.000,E1 98.276} C_DIS
LIN {X 0.099,Y -624.335,Z 1227.344,A 0.000,B 0.000,C 90.000,E1 97.871} C_DIS
LIN {X 0.182,Y -620.734,Z 1227.341,A 0.000,B 0.000,C 90.000,E1 97.352} C_DIS
LIN {X -0.130,Y -618.844,Z 1227.340,A 0.000,B 0.000,C 90.000,E1 97.125} C_DIS
LIN {X -0.171,Y -612.866,Z 1227.336,A 0.000,B 0.000,C 90.000,E1 96.486} C_DIS
LIN {X 0.065,Y -607.439,Z 1227.333,A 0.000,B 0.000,C 90.000,E1 95.967} C_DIS
LIN {X -0.029,Y -603.244,Z 1227.331,A 0.000,B 0.000,C 90.000,E1 95.625} C_DIS
LIN {X 0.056,Y -600.326,Z 1227.330,A 0.000,B 0.000,C 90.000,E1 95.391} C_DIS
LIN {X -0.079,Y -592.611,Z 1227.327,A 0.000,B 0.000,C 90.000,E1 94.878} C_DIS
LIN {X 0.276,Y -584.656,Z 1227.324,A 0.000,B 0.000,C 90.000,E1 94.359} C_DIS
LIN {X 0.094,Y -580.806,Z 1227.323,A 0.000,B 0.000,C 90.000,E1 94.188} C_DIS
LIN {X 0.038,Y -570.895,Z 1227.321,A 0.000,B 0.000,C 90.000,E1 93.726} C_DIS
LIN {X 0.184,Y -567.165,Z 1227.320,A 0.000,B 0.000,C 90.000,E1 93.498} C_DIS
LIN {X -0.096,Y -566.479,Z 1227.319,A 0.000,B 0.000,C 90.000,E1 93.440} C_DIS
LIN {X -0.152,Y -566.459,Z 1227.319,A 0.000,B 0.000,C 90.000,E1 93.440} C_DIS
LIN {X 0.241,Y -566.027,Z 1227.318,A 0.000,B 0.000,C 90.000,E1 93.212} C_DIS
LIN {X 0.264,Y -565.074,Z 1227.316,A 0.000,B 0.000,C 90.000,E1 92.922} C_DIS
LIN {X -0.193,Y -564.974,Z 1227.314,A 0.000,B 0.000,C 90.000,E1 92.522} C_DIS
LIN {X -0.187,Y -565.712,Z 1227.306,A 0.000,B 0.000,C 90.000,E1 91.146} C_DIS
LIN {X -0.062,Y -566.909,Z 1227.297,A 0.000,B 0.000,C 90.000,E1 89.484} C_DIS
LIN {X 0.102,Y -568.068,Z 1227.288,A 0.000,B 0.000,C 90.000,E1 87.822} C_DIS
LIN {X -0.120,Y -569.532,Z 1227.277,A 0.000,B 0.000,C 90.000,E1 85.927} C_DIS
LIN {X 0.039,Y -571.725,Z 1227.264,A 0.000,B 0.000,C 90.000,E1 83.451} C_DIS
LIN {X -0.184,Y -573.259,Z 1227.255,A 0.000,B 0.000,C 90.000,E1 81.837} C_DIS
LIN {X 0.150,Y -574.445,Z 1227.247,A 0.000,B 0.000,C 90.000,E1 80.443} C_DIS
LIN {X -0.063,Y -575.423,Z 1227.240,A 0.000,B 0.000,C 90.000,E1 79.106} C_DIS
LIN {X 0.274,Y -576.624,Z 1227.229,A 0.000,B 0.000,C 90.000,E1 77.173} C_DIS
LIN {X -0.006,Y -577.270,Z 1227.223,A 0.000,B 0.000,C 90.000,E1 76.117} C_DIS
LIN {X -0.138,Y -577.861,Z 1227.217,A 0.000,B 0.000,C 90.000,E1 75.046} C_DIS
LIN {X 0.323,Y -578.765,Z 1227.208,A 0.000,B 0.000,C 90.000,E1 73.378} C_DIS
LIN {X 0.038,Y -579.489,Z 1227.200,A 0.000,B 0.000,C 90.000,E1 72.054} C_DIS
LIN {X 0.153,Y -580.494,Z 1227.191,A 0.000,B 0.000,C 90.000,E1 70.423} C_DIS
LIN {X 0.239,Y -582.246,Z 1227.176,A 0.000,B 0.000,C 90.000,E1 67.720} C_DIS
LIN {X -0.123,Y -583.388,Z 1227.169,A 0.000,B 0.000,C 90.000,E1 66.410} C_DIS
LIN {X 0.061,Y -584.636,Z 1227.161,A 0.000,B 0.000,C 90.000,E1 65.049} C_DIS
LIN {X -0.125,Y -586.540,Z 1227.150,A 0.000,B 0.000,C 90.000,E1 62.922} C_DIS
LIN {X -0.024,Y -588.212,Z 1227.141,A 0.000,B 0.000,C 90.000,E1 61.307} C_DIS
LIN {X -0.117,Y -589.863,Z 1227.132,A 0.000,B 0.000,C 90.000,E1 59.715} C_DIS
LIN {X -0.066,Y -591.243,Z 1227.124,A 0.000,B 0.000,C 90.000,E1 58.377} C_DIS
LIN {X 0.002,Y -592.445,Z 1227.117,A 0.000,B 0.000,C 90.000,E1 57.041} C_DIS
LIN {X -0.088,Y -593.584,Z 1227.110,A 0.000,B 0.000,C 90.000,E1 55.722} C_DIS
LIN {X 0.106,Y -594.406,Z 1227.104,A 0.000,B 0.000,C 90.000,E1 54.642} C_DIS
LIN {X -0.092,Y -595.482,Z 1227.096,A 0.000,B 0.000,C 90.000,E1 53.336} C_DIS
LIN {X 0.202,Y -596.881,Z 1227.086,A 0.000,B 0.000,C 90.000,E1 51.457} C_DIS
LIN {X 0.052,Y -597.449,Z 1227.082,A 0.000,B 0.000,C 90.000,E1 50.678} C_DIS
LIN {X -0.167,Y -598.240,Z 1227.071,A 0.000,B 0.000,C 90.000,E1 48.852} C_DIS
LIN {X 0.033,Y -598.865,Z 1227.064,A 0.000,B 0.000,C 90.000,E1 47.514} C_DIS
LIN {X 0.050,Y -599.137,Z 1227.058,A 0.000,B 0.000,C 90.000,E1 46.458} C_DIS
LIN {X -0.168,Y -599.244,Z 1227.051,A 0.000,B 0.000,C 90.000,E1 45.162} C_DIS
LIN {X -0.171,Y -599.112,Z 1227.045,A 0.000,B 0.000,C 90.000,E1 44.109} C_DIS
LIN {X 0.257,Y -598.787,Z 1227.039,A 0.000,B 0.000,C 90.000,E1 43.014} C_DIS
LIN {X 0.052,Y -598.444,Z 1227.035,A 0.000,B 0.000,C 90.000,E1 42.243} C_DIS
LIN {X 0.248,Y -597.453,Z 1227.025,A 0.000,B 0.000,C 90.000,E1 40.378} C_DIS
LIN {X -0.132,Y -596.844,Z 1227.019,A 0.000,B 0.000,C 90.000,E1 39.358} C_DIS
LIN {X 0.096,Y -596.220,Z 1227.014,A 0.000,B 0.000,C 90.000,E1 38.543} C_DIS
LIN {X -0.067,Y -594.897,Z 1227.007,A 0.000,B 0.000,C 90.000,E1 37.237} C_DIS
LIN {X 0.130,Y -593.913,Z 1227.002,A 0.000,B 0.000,C 90.000,E1 36.423} C_DIS
LIN {X -0.168,Y -592.407,Z 1226.997,A 0.000,B 0.000,C 90.000,E1 35.391} C_DIS
LIN {X -0.143,Y -590.465,Z 1226.991,A 0.000,B 0.000,C 90.000,E1 34.326} C_DIS
LIN {X -0.064,Y -589.353,Z 1226.988,A 0.000,B 0.000,C 90.000,E1 33.785} C_DIS
LIN {X 0.207,Y -587.448,Z 1226.983,A 0.000,B 0.000,C 90.000,E1 32.959} C_DIS
LIN {X -0.355,Y -585.394,Z 1226.979,A 0.000,B 0.000,C 90.000,E1 32.212} C_DIS
LIN {X -0.134,Y -582.827,Z 1226.974,A 0.000,B 0.000,C 90.000,E1 31.386} C_DIS
LIN {X -0.106,Y -580.960,Z 1226.971,A 0.000,B 0.000,C 90.000,E1 30.846} C_DIS
LIN {X 0.263,Y -577.730,Z 1226.967,A 0.000,B 0.000,C 90.000,E1 30.001} C_DIS
LIN {X 0.099,Y -574.169,Z 1226.962,A 0.000,B 0.000,C 90.000,E1 29.205} C_DIS
LIN {X -0.215,Y -571.442,Z 1226.959,A 0.000,B 0.000,C 90.000,E1 28.693} C_DIS
LIN {X -0.037,Y -566.244,Z 1226.954,A 0.000,B 0.000,C 90.000,E1 27.719} C_DIS
LIN {X -0.048,Y -563.891,Z 1226.952,A 0.000,B 0.000,C 90.000,E1 27.308} C_DIS
LIN {X 0.072,Y -560.497,Z 1226.949,A 0.000,B 0.000,C 90.000,E1 26.744} C_DIS
LIN {X 0.172,Y -556.886,Z 1226.946,A 0.000,B 0.000,C 90.000,E1 26.181} C_DIS
LIN {X -0.010,Y -553.043,Z 1226.943,A 0.000,B 0.000,C 90.000,E1 25.643} C_DIS
LIN {X 0.037,Y -548.919,Z 1226.939,A 0.000,B 0.000,C 90.000,E1 25.079} C_DIS
LIN {X -0.069,Y -543.270,Z 1226.936,A 0.000,B 0.000,C 90.000,E1 24.387} C_DIS
LIN {X 0.084,Y -538.707,Z 1226.932,A 0.000,B 0.000,C 90.000,E1 23.823} C_DIS
LIN {X 0.314,Y -531.291,Z 1226.928,A 0.000,B 0.000,C 90.000,E1 22.950} C_DIS
LIN {X -0.260,Y -522.148,Z 1226.922,A 0.000,B 0.000,C 90.000,E1 22.025} C_DIS
LIN {X -0.264,Y -511.334,Z 1226.916,A 0.000,B 0.000,C 90.000,E1 20.918} C_DIS
LIN {X -0.088,Y -500.212,Z 1226.910,A 0.000,B 0.000,C 90.000,E1 19.812} C_DIS
LIN {X 0.190,Y -490.367,Z 1226.905,A 0.000,B 0.000,C 90.000,E1 18.852} C_DIS
LIN {X -0.165,Y -483.071,Z 1226.901,A 0.000,B 0.000,C 90.000,E1 18.236} C_DIS
LIN {X 0.018,Y -469.761,Z 1226.895,A 0.000,B 0.000,C 90.000,E1 17.040} C_DIS
LIN {X -0.213,Y -453.519,Z 1226.887,A 0.000,B 0.000,C 90.000,E1 15.607} C_DIS
LIN {X 0.130,Y -430.508,Z 1226.874,A 0.000,B 0.000,C 90.000,E1 13.355} C_DIS
LIN {X -0.134,Y -410.556,Z 1226.862,A 0.000,B 0.000,C 90.000,E1 11.243} C_DIS
LIN {X 0.080,Y -402.381,Z 1226.857,A 0.000,B 0.000,C 90.000,E1 10.254} C_DIS
LIN {X 0.142,Y -398.427,Z 1226.854,A 0.000,B 0.000,C 90.000,E1 9.726} C_DIS
LIN {X 0.088,Y -395.093,Z 1226.851,A 0.000,B 0.000,C 90.000,E1 9.208} C_DIS
LIN {X -0.130,Y -393.959,Z 1226.849,A 0.000,B 0.000,C 90.000,E1 8.916} C_DIS
LIN {X -0.168,Y -393.950,Z 1226.849,A 0.000,B 0.000,C 90.000,E1 8.916} C_DIS
LIN {X 0.082,Y -393.996,Z 1226.848,A 0.000,B 0.000,C 90.000,E1 8.681} C_DIS
LIN {X 0.044,Y -394.012,Z 1226.848,A 0.000,B 0.000,C 90.000,E1 8.681} C_DIS
LIN {X 0.093,Y -396.775,Z 1226.845,A 0.000,B 0.000,C 90.000,E1 8.049} C_DIS
LIN {X 0.012,Y -400.362,Z 1226.843,A 0.000,B 0.000,C 90.000,E1 7.644} C_DIS
LIN {X -0.190,Y -404.251,Z 1226.841,A 0.000,B 0.000,C 90.000,E1 7.352} C_DIS
LIN {X 0.171,Y -418.902,Z 1226.835,A 0.000,B 0.000,C 90.000,E1 6.201} C_DIS
LIN {X 0.206,Y -433.270,Z 1226.829,A 0.000,B 0.000,C 90.000,E1 5.106} C_DIS
LIN {X 0.197,Y -445.925,Z 1226.823,A 0.000,B 0.000,C 90.000,E1 4.131} C_DIS
LIN {X 0.220,Y -460.092,Z 1226.817,A 0.000,B 0.000,C 90.000,E1 3.037} C_DIS
LIN {X -0.055,Y -467.717,Z 1226.814,A 0.000,B 0.000,C 90.000,E1 2.465} C_DIS
LIN {X 0.153,Y -472.296,Z 1226.812,A 0.000,B 0.000,C 90.000,E1 2.064} C_DIS
LIN {X 0.004,Y -479.521,Z 1226.808,A 0.000,B 0.000,C 90.000,E1 1.432} C_DIS
LIN {X 0.226,Y -485.246,Z 1226.805,A 0.000,B 0.000,C 90.000,E1 0.859} C_DIS
LIN {X 0.124,Y -492.021,Z 1226.801,A 0.000,B 0.000,C 90.000,E1 0.172} C_DIS
LIN {X 0.148,Y -498.212,Z 1226.797,A 0.000,B 0.000,C 90.000,E1 359.484} C_DIS
LIN {X 0.215,Y -504.313,Z 1226.793,A 0.000,B 0.000,C 90.000,E1 358.740} C_DIS
LIN {X -0.182,Y -509.935,Z 1226.789,A 0.000,B 0.000,C 90.000,E1 358.051} C_DIS
LIN {X -0.147,Y -515.157,Z 1226.785,A 0.000,B 0.000,C 90.000,E1 357.306} C_DIS
LIN {X -0.043,Y -520.042,Z 1226.781,A 0.000,B 0.000,C 90.000,E1 356.560} C_DIS
LIN {X -0.161,Y -523.683,Z 1226.778,A 0.000,B 0.000,C 90.000,E1 355.988} C_DIS
LIN {X 0.024,Y -527.811,Z 1226.774,A 0.000,B 0.000,C 90.000,E1 355.241} C_DIS
LIN {X -0.231,Y -531.544,Z 1226.770,A 0.000,B 0.000,C 90.000,E1 354.546} C_DIS
LIN {X -0.226,Y -534.341,Z 1226.766,A 0.000,B 0.000,C 90.000,E1 353.970} C_DIS
LIN {X -0.200,Y -536.911,Z 1226.763,A 0.000,B 0.000,C 90.000,E1 353.394} C_DIS
LIN {X -0.097,Y -540.404,Z 1226.758,A 0.000,B 0.000,C 90.000,E1 352.527} C_DIS
LIN {X -0.034,Y -542.594,Z 1226.755,A 0.000,B 0.000,C 90.000,E1 351.951} C_DIS
LIN {X 0.125,Y -545.563,Z 1226.751,A 0.000,B 0.000,C 90.000,E1 351.084} C_DIS
LIN {X -0.228,Y -548.272,Z 1226.746,A 0.000,B 0.000,C 90.000,E1 350.274} C_DIS
LIN {X 0.190,Y -551.439,Z 1226.740,A 0.000,B 0.000,C 90.000,E1 349.106} C_DIS
LIN {X 0.246,Y -555.089,Z 1226.732,A 0.000,B 0.000,C 90.000,E1 347.701} C_DIS
LIN {X 0.090,Y -557.027,Z 1226.727,A 0.000,B 0.000,C 90.000,E1 346.881} C_DIS
LIN {X -0.175,Y -559.975,Z 1226.719,A 0.000,B 0.000,C 90.000,E1 345.519} C_DIS
LIN {X -0.141,Y -561.631,Z 1226.715,A 0.000,B 0.000,C 90.000,E1 344.685} C_DIS
LIN {X 0.062,Y -563.609,Z 1226.709,A 0.000,B 0.000,C 90.000,E1 343.559} C_DIS
LIN {X 0.064,Y -565.781,Z 1226.701,A 0.000,B 0.000,C 90.000,E1 342.181} C_DIS
LIN {X 0.279,Y -567.575,Z 1226.693,A 0.000,B 0.000,C 90.000,E1 340.786} C_DIS
LIN {X -0.158,Y -568.452,Z 1226.689,A 0.000,B 0.000,C 90.000,E1 340.007} C_DIS
LIN {X 0.136,Y -569.076,Z 1226.684,A 0.000,B 0.000,C 90.000,E1 339.156} C_DIS
LIN {X 0.113,Y -569.482,Z 1226.680,A 0.000,B 0.000,C 90.000,E1 338.337} C_DIS
LIN {X -0.111,Y -569.624,Z 1226.675,A 0.000,B 0.000,C 90.000,E1 337.539} C_DIS
LIN {X 0.006,Y -569.219,Z 1226.669,A 0.000,B 0.000,C 90.000,E1 336.433} C_DIS
LIN {X -0.004,Y -568.536,Z 1226.665,A 0.000,B 0.000,C 90.000,E1 335.613} C_DIS
LIN {X -0.019,Y -567.563,Z 1226.660,A 0.000,B 0.000,C 90.000,E1 334.793} C_DIS
LIN {X -0.047,Y -566.171,Z 1226.655,A 0.000,B 0.000,C 90.000,E1 333.973} C_DIS
LIN {X -0.159,Y -565.071,Z 1226.652,A 0.000,B 0.000,C 90.000,E1 333.435} C_DIS
LIN {X 0.095,Y -562.380,Z 1226.646,A 0.000,B 0.000,C 90.000,E1 332.308} C_DIS
LIN {X -0.230,Y -559.909,Z 1226.642,A 0.000,B 0.000,C 90.000,E1 331.513} C_DIS
LIN {X 0.328,Y -558.931,Z 1226.640,A 0.000,B 0.000,C 90.000,E1 331.179} C_DIS
LIN {X -0.085,Y -556.650,Z 1226.637,A 0.000,B 0.000,C 90.000,E1 330.667} C_DIS
LIN {X 0.129,Y -553.464,Z 1226.633,A 0.000,B 0.000,C 90.000,E1 329.950} C_DIS
LIN {X 0.066,Y -551.310,Z 1226.631,A 0.000,B 0.000,C 90.000,E1 329.537} C_DIS
LIN {X -0.124,Y -548.114,Z 1226.628,A 0.000,B 0.000,C 90.000,E1 328.997} C_DIS
LIN {X 0.131,Y -544.647,Z 1226.625,A 0.000,B 0.000,C 90.000,E1 328.408} C_DIS
LIN {X 0.048,Y -539.915,Z 1226.621,A 0.000,B 0.000,C 90.000,E1 327.709} C_DIS
LIN {X 0.235,Y -535.828,Z 1226.618,A 0.000,B 0.000,C 90.000,E1 327.120} C_DIS
LIN {X 0.102,Y -528.083,Z 1226.612,A 0.000,B 0.000,C 90.000,E1 326.135} C_DIS
LIN {X 0.047,Y -516.790,Z 1226.604,A 0.000,B 0.000,C 90.000,E1 324.689} C_DIS
LIN {X -0.193,Y -513.458,Z 1226.601,A 0.000,B 0.000,C 90.000,E1 324.196} C_DIS
LIN {X -0.242,Y -510.848,Z 1226.598,A 0.000,B 0.000,C 90.000,E1 323.703} C_DIS
LIN {X -0.002,Y -508.870,Z 1226.595,A 0.000,B 0.000,C 90.000,E1 323.084} C_DIS
LIN {X -0.153,Y -508.164,Z 1226.592,A 0.000,B 0.000,C 90.000,E1 322.637} C_DIS
LIN {X 0.064,Y -507.611,Z 1226.591,A 0.000,B 0.000,C 90.000,E1 322.316} C_DIS
LIN {X -0.093,Y -506.993,Z 1226.586,A 0.000,B 0.000,C 90.000,E1 321.457} C_DIS
LIN {X -0.073,Y -506.991,Z 1226.581,A 0.000,B 0.000,C 90.000,E1 320.561} C_DIS
LIN {X -0.003,Y -508.465,Z 1226.566,A 0.000,B 0.000,C 90.000,E1 317.877} C_DIS
LIN {X -0.116,Y -509.128,Z 1226.559,A 0.000,B 0.000,C 90.000,E1 316.701} C_DIS
LIN {X 0.022,Y -509.796,Z 1226.551,A 0.000,B 0.000,C 90.000,E1 315.202} C_DIS
LIN {X 0.068,Y -510.473,Z 1226.541,A 0.000,B 0.000,C 90.000,E1 313.419} C_DIS
LIN {X 0.240,Y -511.164,Z 1226.533,A 0.000,B 0.000,C 90.000,E1 311.919} C_DIS
LIN {X 0.075,Y -511.805,Z 1226.525,A 0.000,B 0.000,C 90.000,E1 310.458} C_DIS
LIN {X -0.018,Y -512.357,Z 1226.517,A 0.000,B 0.000,C 90.000,E1 308.991} C_DIS
LIN {X -0.177,Y -512.898,Z 1226.507,A 0.000,B 0.000,C 90.000,E1 307.237} C_DIS
LIN {X 0.152,Y -513.369,Z 1226.499,A 0.000,B 0.000,C 90.000,E1 305.724} C_DIS
LIN {X -0.182,Y -513.950,Z 1226.489,A 0.000,B 0.000,C 90.000,E1 303.992} C_DIS
LIN {X 0.005,Y -514.363,Z 1226.481,A 0.000,B 0.000,C 90.000,E1 302.498} C_DIS
LIN {X 0.201,Y -514.580,Z 1226.472,A 0.000,B 0.000,C 90.000,E1 301.003} C_DIS
LIN {X 0.128,Y -514.750,Z 1226.464,A 0.000,B 0.000,C 90.000,E1 299.539} C_DIS
LIN {X 0.148,Y -514.846,Z 1226.458,A 0.000,B 0.000,C 90.000,E1 298.359} C_DIS
LIN {X 0.280,Y -514.962,Z 1226.449,A 0.000,B 0.000,C 90.000,E1 296.873} C_DIS
LIN {X 0.306,Y -515.059,Z 1226.436,A 0.000,B 0.000,C 90.000,E1 294.515} C_DIS
LIN {X -0.132,Y -515.132,Z 1226.430,A 0.000,B 0.000,C 90.000,E1 293.387} C_DIS
LIN {X -0.096,Y -515.122,Z 1226.423,A 0.000,B 0.000,C 90.000,E1 292.206} C_DIS
LIN {X 0.003,Y -514.555,Z 1226.414,A 0.000,B 0.000,C 90.000,E1 290.429} C_DIS
LIN {X -0.082,Y -513.686,Z 1226.404,A 0.000,B 0.000,C 90.000,E1 288.671} C_DIS
LIN {X 0.188,Y -513.028,Z 1226.396,A 0.000,B 0.000,C 90.000,E1 287.166} C_DIS
LIN {X -0.127,Y -512.062,Z 1226.384,A 0.000,B 0.000,C 90.000,E1 285.134} C_DIS
LIN {X -0.114,Y -510.804,Z 1226.373,A 0.000,B 0.000,C 90.000,E1 283.063} C_DIS
LIN {X 0.276,Y -509.589,Z 1226.363,A 0.000,B 0.000,C 90.000,E1 281.243} C_DIS
LIN {X -0.059,Y -508.284,Z 1226.353,A 0.000,B 0.000,C 90.000,E1 279.500} C_DIS
LIN {X -0.196,Y -507.703,Z 1226.348,A 0.000,B 0.000,C 90.000,E1 278.624} C_DIS
LIN {X 0.184,Y -506.204,Z 1226.335,A 0.000,B 0.000,C 90.000,E1 276.201} C_DIS
LIN {X -0.036,Y -504.902,Z 1226.321,A 0.000,B 0.000,C 90.000,E1 273.841} C_DIS
LIN {X 0.053,Y -504.173,Z 1226.315,A 0.000,B 0.000,C 90.000,E1 272.636} C_DIS
LIN {X 0.132,Y -503.372,Z 1226.308,A 0.000,B 0.000,C 90.000,E1 271.432} C_DIS
LIN {X 0.110,Y -501.626,Z 1226.293,A 0.000,B 0.000,C 90.000,E1 268.740} C_DIS
LIN {X 0.029,Y -500.772,Z 1226.285,A 0.000,B 0.000,C 90.000,E1 267.249} C_DIS
LIN {X 0.055,Y -500.109,Z 1226.278,A 0.000,B 0.000,C 90.000,E1 266.045} C_DIS
LIN {X -0.118,Y -498.919,Z 1226.268,A 0.000,B 0.000,C 90.000,E1 264.261} C_DIS
LIN {X -0.085,Y -497.965,Z 1226.261,A 0.000,B 0.000,C 90.000,E1 263.053} C_DIS
LIN {X -0.180,Y -496.255,Z 1226.251,A 0.000,B 0.000,C 90.000,E1 261.254} C_DIS
LIN {X -0.215,Y -494.932,Z 1226.243,A 0.000,B 0.000,C 90.000,E1 259.746} C_DIS
LIN {X 0.097,Y -493.126,Z 1226.231,A 0.000,B 0.000,C 90.000,E1 257.589} C_DIS
LIN {X 0.093,Y -491.630,Z 1226.219,A 0.000,B 0.000,C 90.000,E1 255.463} C_DIS
LIN {X 0.179,Y -490.297,Z 1226.208,A 0.000,B 0.000,C 90.000,E1 253.323} C_DIS
LIN {X -0.101,Y -489.254,Z 1226.196,A 0.000,B 0.000,C 90.000,E1 251.221} C_DIS
LIN {X -0.114,Y -488.368,Z 1226.185,A 0.000,B 0.000,C 90.000,E1 249.390} C_DIS
LIN {X 0.007,Y -487.535,Z 1226.177,A 0.000,B 0.000,C 90.000,E1 247.847} C_DIS
LIN {X 0.107,Y -486.465,Z 1226.168,A 0.000,B 0.000,C 90.000,E1 246.305} C_DIS
LIN {X 0.148,Y -484.936,Z 1226.158,A 0.000,B 0.000,C 90.000,E1 244.460} C_DIS
LIN {X 0.156,Y -483.270,Z 1226.148,A 0.000,B 0.000,C 90.000,E1 242.615} C_DIS
LIN {X -0.067,Y -481.774,Z 1226.139,A 0.000,B 0.000,C 90.000,E1 241.101} C_DIS
LIN {X -0.107,Y -480.430,Z 1226.133,A 0.000,B 0.000,C 90.000,E1 239.871} C_DIS
LIN {X 0.062,Y -478.362,Z 1226.122,A 0.000,B 0.000,C 90.000,E1 237.995} C_DIS
LIN {X 0.244,Y -476.616,Z 1226.114,A 0.000,B 0.000,C 90.000,E1 236.421} C_DIS
LIN {X -0.034,Y -474.243,Z 1226.102,A 0.000,B 0.000,C 90.000,E1 234.276} C_DIS
LIN {X -0.201,Y -471.956,Z 1226.089,A 0.000,B 0.000,C 90.000,E1 232.110} C_DIS
LIN {X -0.058,Y -469.627,Z 1226.075,A 0.000,B 0.000,C 90.000,E1 229.585} C_DIS
LIN {X -0.019,Y -468.582,Z 1226.068,A 0.000,B 0.000,C 90.000,E1 228.324} C_DIS
LIN {X -0.213,Y -466.922,Z 1226.058,A 0.000,B 0.000,C 90.000,E1 226.458} C_DIS
LIN {X -0.117,Y -463.986,Z 1226.021,A 0.000,B 0.000,C 90.000,E1 219.806} C_DIS
LIN {X -0.159,Y -465.037,Z 1226.000,A 0.000,B 0.000,C 90.000,E1 216.011} C_DIS
LIN {X -0.064,Y -466.113,Z 1225.988,A 0.000,B 0.000,C 90.000,E1 213.785} C_DIS
LIN {X 0.271,Y -468.818,Z 1225.970,A 0.000,B 0.000,C 90.000,E1 210.590} C_DIS
LIN {X 0.176,Y -472.231,Z 1225.953,A 0.000,B 0.000,C 90.000,E1 207.462} C_DIS
LIN {X 0.098,Y -474.930,Z 1225.941,A 0.000,B 0.000,C 90.000,E1 205.283} C_DIS
LIN {X -0.191,Y -480.577,Z 1225.920,A 0.000,B 0.000,C 90.000,E1 201.589} C_DIS
LIN {X 0.084,Y -484.568,Z 1225.908,A 0.000,B 0.000,C 90.000,E1 199.396} C_DIS
LIN {X -0.148,Y -489.129,Z 1225.896,A 0.000,B 0.000,C 90.000,E1 197.275} C_DIS
LIN {X -0.055,Y -494.912,Z 1225.882,A 0.000,B 0.000,C 90.000,E1 194.828} C_DIS
LIN {X 0.087,Y -498.860,Z 1225.874,A 0.000,B 0.000,C 90.000,E1 193.300} C_DIS
LIN {X -0.183,Y -502.902,Z 1225.866,A 0.000,B 0.000,C 90.000,E1 191.827} C_DIS
LIN {X -0.095,Y -508.660,Z 1225.854,A 0.000,B 0.000,C 90.000,E1 189.726} C_DIS
LIN {X 0.118,Y -513.016,Z 1225.846,A 0.000,B 0.000,C 90.000,E1 188.219} C_DIS
LIN {X -0.164,Y -517.283,Z 1225.838,A 0.000,B 0.000,C 90.000,E1 186.777} C_DIS
LIN {X 0.161,Y -520.646,Z 1225.831,A 0.000,B 0.000,C 90.000,E1 185.568} C_DIS
LIN {X -0.038,Y -525.631,Z 1225.821,A 0.000,B 0.000,C 90.000,E1 183.841} C_DIS
LIN {X -0.199,Y -530.707,Z 1225.812,A 0.000,B 0.000,C 90.000,E1 182.121} C_DIS
LIN {X -0.250,Y -535.603,Z 1225.802,A 0.000,B 0.000,C 90.000,E1 180.401} C_DIS
LIN {X -0.231,Y -538.866,Z 1225.796,A 0.000,B 0.000,C 90.000,E1 179.255} C_DIS
LIN {X -0.130,Y -542.817,Z 1225.788,A 0.000,B 0.000,C 90.000,E1 177.822} C_DIS
LIN {X -0.049,Y -545.108,Z 1225.783,A 0.000,B 0.000,C 90.000,E1 176.963} C_DIS
LIN {X 0.195,Y -548.784,Z 1225.775,A 0.000,B 0.000,C 90.000,E1 175.527} C_DIS
LIN {X -0.181,Y -550.941,Z 1225.771,A 0.000,B 0.000,C 90.000,E1 174.723} C_DIS
LIN {X 0.115,Y -553.762,Z 1225.764,A 0.000,B 0.000,C 90.000,E1 173.571} C_DIS
LIN {X 0.153,Y -557.860,Z 1225.755,A 0.000,B 0.000,C 90.000,E1 171.894} C_DIS
LIN {X -0.127,Y -562.561,Z 1225.744,A 0.000,B 0.000,C 90.000,E1 169.982} C_DIS
LIN {X 0.293,Y -566.460,Z 1225.735,A 0.000,B 0.000,C 90.000,E1 168.285} C_DIS
LIN {X -0.126,Y -571.138,Z 1225.724,A 0.000,B 0.000,C 90.000,E1 166.408} C_DIS
LIN {X -0.306,Y -575.936,Z 1225.714,A 0.000,B 0.000,C 90.000,E1 164.519} C_DIS
LIN {X 0.048,Y -584.333,Z 1225.697,A 0.000,B 0.000,C 90.000,E1 161.511} C_DIS
LIN {X 0.282,Y -595.528,Z 1225.680,A 0.000,B 0.000,C 90.000,E1 158.284} C_DIS
LIN {X 0.156,Y -600.775,Z 1225.672,A 0.000,B 0.000,C 90.000,E1 156.975} C_DIS
LIN {X 0.009,Y -608.052,Z 1225.662,A 0.000,B 0.000,C 90.000,E1 155.153} C_DIS
LIN {X 0.120,Y -611.976,Z 1225.656,A 0.000,B 0.000,C 90.000,E1 154.101} C_DIS
LIN {X -0.034,Y -616.813,Z 1225.649,A 0.000,B 0.000,C 90.000,E1 152.820} C_DIS
LIN {X 0.181,Y -621.326,Z 1225.642,A 0.000,B 0.000,C 90.000,E1 151.513} C_DIS
LIN {X -0.068,Y -624.925,Z 1225.636,A 0.000,B 0.000,C 90.000,E1 150.511} C_DIS
LIN {X -0.231,Y -630.205,Z 1225.628,A 0.000,B 0.000,C 90.000,E1 148.997} C_DIS
LIN {X 0.000,Y -634.474,Z 1225.621,A 0.000,B 0.000,C 90.000,E1 147.709} C_DIS
LIN {X -0.078,Y -637.658,Z 1225.615,A 0.000,B 0.000,C 90.000,E1 146.707} C_DIS
LIN {X -0.161,Y -640.018,Z 1225.611,A 0.000,B 0.000,C 90.000,E1 145.960} C_DIS
LIN {X 0.138,Y -642.267,Z 1225.607,A 0.000,B 0.000,C 90.000,E1 145.182} C_DIS
LIN {X 0.400,Y -645.651,Z 1225.600,A 0.000,B 0.000,C 90.000,E1 143.909} C_DIS
LIN {X -0.140,Y -647.537,Z 1225.596,A 0.000,B 0.000,C 90.000,E1 143.210} C_DIS
LIN {X 0.121,Y -651.060,Z 1225.587,A 0.000,B 0.000,C 90.000,E1 141.698} C_DIS
LIN {X -0.095,Y -653.922,Z 1225.580,A 0.000,B 0.000,C 90.000,E1 140.481} C_DIS
LIN {X 0.291,Y -656.100,Z 1225.575,A 0.000,B 0.000,C 90.000,E1 139.461} C_DIS
LIN {X 0.108,Y -659.942,Z 1225.565,A 0.000,B 0.000,C 90.000,E1 137.757} C_DIS
LIN {X 0.041,Y -662.631,Z 1225.559,A 0.000,B 0.000,C 90.000,E1 136.539} C_DIS
LIN {X -0.020,Y -667.858,Z 1225.546,A 0.000,B 0.000,C 90.000,E1 134.352} C_DIS
LIN {X 0.084,Y -672.735,Z 1225.536,A 0.000,B 0.000,C 90.000,E1 132.405} C_DIS
LIN {X 0.157,Y -675.195,Z 1225.530,A 0.000,B 0.000,C 90.000,E1 131.434} C_DIS
LIN {X -0.047,Y -679.415,Z 1225.521,A 0.000,B 0.000,C 90.000,E1 129.769} C_DIS
LIN {X -0.095,Y -683.035,Z 1225.513,A 0.000,B 0.000,C 90.000,E1 128.338} C_DIS
LIN {X 0.360,Y -686.646,Z 1225.505,A 0.000,B 0.000,C 90.000,E1 126.870} C_DIS
LIN {X 0.236,Y -688.974,Z 1225.500,A 0.000,B 0.000,C 90.000,E1 125.931} C_DIS
LIN {X -0.027,Y -692.223,Z 1225.492,A 0.000,B 0.000,C 90.000,E1 124.532} C_DIS
LIN {X -0.265,Y -694.862,Z 1225.485,A 0.000,B 0.000,C 90.000,E1 123.372} C_DIS
LIN {X -0.113,Y -696.923,Z 1225.480,A 0.000,B 0.000,C 90.000,E1 122.418} C_DIS
LIN {X 0.064,Y -698.779,Z 1225.475,A 0.000,B 0.000,C 90.000,E1 121.465} C_DIS
LIN {X -0.438,Y -701.063,Z 1225.468,A 0.000,B 0.000,C 90.000,E1 120.335} C_DIS
LIN {X 0.048,Y -703.171,Z 1225.462,A 0.000,B 0.000,C 90.000,E1 119.127} C_DIS
LIN {X -0.403,Y -704.602,Z 1225.457,A 0.000,B 0.000,C 90.000,E1 118.231} C_DIS
LIN {X -0.166,Y -705.402,Z 1225.453,A 0.000,B 0.000,C 90.000,E1 117.513} C_DIS
LIN {X 0.051,Y -706.073,Z 1225.448,A 0.000,B 0.000,C 90.000,E1 116.565} C_DIS
LIN {X 0.298,Y -706.362,Z 1225.444,A 0.000,B 0.000,C 90.000,E1 115.848} C_DIS
LIN {X 0.237,Y -706.322,Z 1225.440,A 0.000,B 0.000,C 90.000,E1 115.155} C_DIS
LIN {X 0.178,Y -705.796,Z 1225.436,A 0.000,B 0.000,C 90.000,E1 114.463} C_DIS
LIN {X -0.174,Y -704.898,Z 1225.433,A 0.000,B 0.000,C 90.000,E1 114.027} C_DIS
LIN {X 0.113,Y -704.077,Z 1225.432,A 0.000,B 0.000,C 90.000,E1 113.770} C_DIS
LIN {X -0.246,Y -701.956,Z 1225.430,A 0.000,B 0.000,C 90.000,E1 113.334} C_DIS
LIN {X -0.108,Y -701.107,Z 1225.429,A 0.000,B 0.000,C 90.000,E1 113.206} C_DIS
LIN {X 0.030,Y -699.874,Z 1225.428,A 0.000,B 0.000,C 90.000,E1 113.078} C_DIS
LIN {X 0.321,Y -694.897,Z 1225.426,A 0.000,B 0.000,C 90.000,E1 112.642} C_DIS
LIN {X -0.346,Y -692.853,Z 1225.425,A 0.000,B 0.000,C 90.000,E1 112.589} C_DIS
LIN {X 0.071,Y -686.026,Z 1225.424,A 0.000,B 0.000,C 90.000,E1 112.333} C_DIS
LIN {X -0.180,Y -684.864,Z 1225.424,A 0.000,B 0.000,C 90.000,E1 112.333} C_DIS
LIN {X -0.030,Y -677.212,Z 1225.424,A 0.000,B 0.000,C 90.000,E1 112.280} C_DIS
LIN {X -0.060,Y -615.170,Z 1225.424,A 0.000,B 0.000,C 90.000,E1 112.280} C_DIS
LIN {X -0.035,Y -612.775,Z 1225.423,A 0.000,B 0.000,C 90.000,E1 112.153} C_DIS
LIN {X 0.196,Y -609.655,Z 1225.422,A 0.000,B 0.000,C 90.000,E1 111.897} C_DIS
LIN {X 0.170,Y -609.024,Z 1225.422,A 0.000,B 0.000,C 90.000,E1 111.844} C_DIS
LIN {X 0.319,Y -607.170,Z 1225.420,A 0.000,B 0.000,C 90.000,E1 111.589} C_DIS
LIN {X -0.150,Y -606.426,Z 1225.420,A 0.000,B 0.000,C 90.000,E1 111.535} C_DIS
LIN {X -0.180,Y -606.441,Z 1225.418,A 0.000,B 0.000,C 90.000,E1 111.334} C_DIS
LIN {X 0.133,Y -606.668,Z 1225.418,A 0.000,B 0.000,C 90.000,E1 111.173} C_DIS
LIN {X 0.333,Y -609.103,Z 1225.414,A 0.000,B 0.000,C 90.000,E1 110.482} C_DIS
LIN {X 0.258,Y -613.588,Z 1225.408,A 0.000,B 0.000,C 90.000,E1 109.450} C_DIS
LIN {X -0.297,Y -616.370,Z 1225.404,A 0.000,B 0.000,C 90.000,E1 108.725} C_DIS
LIN {X 0.308,Y -620.104,Z 1225.398,A 0.000,B 0.000,C 90.000,E1 107.638} C_DIS
LIN {X -0.025,Y -625.208,Z 1225.391,A 0.000,B 0.000,C 90.000,E1 106.386} C_DIS
LIN {X 0.127,Y -628.020,Z 1225.387,A 0.000,B 0.000,C 90.000,E1 105.607} C_DIS
LIN {X -0.074,Y -628.951,Z 1225.385,A 0.000,B 0.000,C 90.000,E1 105.371} C_DIS
LIN {X 0.304,Y -630.519,Z 1225.383,A 0.000,B 0.000,C 90.000,E1 104.828} C_DIS
LIN {X -0.270,Y -632.446,Z 1225.378,A 0.000,B 0.000,C 90.000,E1 104.120} C_DIS
LIN {X -0.029,Y -633.436,Z 1225.375,A 0.000,B 0.000,C 90.000,E1 103.592} C_DIS
LIN {X 0.043,Y -634.490,Z 1225.371,A 0.000,B 0.000,C 90.000,E1 102.827} C_DIS
LIN {X 0.304,Y -634.758,Z 1225.369,A 0.000,B 0.000,C 90.000,E1 102.299} C_DIS
LIN {X -0.055,Y -634.636,Z 1225.366,A 0.000,B 0.000,C 90.000,E1 101.827} C_DIS
LIN {X -0.235,Y -634.445,Z 1225.364,A 0.000,B 0.000,C 90.000,E1 101.591} C_DIS
LIN {X -0.100,Y -633.724,Z 1225.362,A 0.000,B 0.000,C 90.000,E1 101.074} C_DIS
LIN {X -0.032,Y -632.039,Z 1225.357,A 0.000,B 0.000,C 90.000,E1 100.310} C_DIS
LIN {X 0.099,Y -630.625,Z 1225.354,A 0.000,B 0.000,C 90.000,E1 99.792} C_DIS
LIN {X -0.292,Y -628.749,Z 1225.352,A 0.000,B 0.000,C 90.000,E1 99.321} C_DIS
LIN {X -0.235,Y -625.659,Z 1225.348,A 0.000,B 0.000,C 90.000,E1 98.681} C_DIS
LIN {X 0.013,Y -623.616,Z 1225.346,A 0.000,B 0.000,C 90.000,E1 98.276} C_DIS
LIN {X 0.090,Y -620.204,Z 1225.343,A 0.000,B 0.000,C 90.000,E1 97.757} C_DIS
LIN {X -0.016,Y -615.069,Z 1225.340,A 0.000,B 0.000,C 90.000,E1 97.125} C_DIS
LIN {X 0.009,Y -610.302,Z 1225.337,A 0.000,B 0.000,C 90.000,E1 96.606} C_DIS
LIN {X -0.316,Y -604.910,Z 1225.334,A 0.000,B 0.000,C 90.000,E1 96.144} C_DIS
LIN {X -0.299,Y -597.733,Z 1225.331,A 0.000,B 0.000,C 90.000,E1 95.568} C_DIS
LIN {X 0.198,Y -589.866,Z 1225.328,A 0.000,B 0.000,C 90.000,E1 94.992} C_DIS
LIN {X -0.201,Y -583.262,Z 1225.326,A 0.000,B 0.000,C 90.000,E1 94.645} C_DIS
LIN {X 0.038,Y -578.236,Z 1225.324,A 0.000,B 0.000,C 90.000,E1 94.359} C_DIS
LIN {X -0.201,Y -571.415,Z 1225.323,A 0.000,B 0.000,C 90.000,E1 94.073} C_DIS
LIN {X -0.197,Y -567.600,Z 1225.321,A 0.000,B 0.000,C 90.000,E1 93.841} C_DIS
LIN {X -0.246,Y -567.523,Z 1225.321,A 0.000,B 0.000,C 90.000,E1 93.841} C_DIS
LIN {X 0.230,Y -565.410,Z 1225.319,A 0.000,B 0.000,C 90.000,E1 93.440} C_DIS
LIN {X 0.188,Y -565.383,Z 1225.319,A 0.000,B 0.000,C 90.000,E1 93.440} C_DIS
LIN {X -0.179,Y -565.078,Z 1225.318,A 0.000,B 0.000,C 90.000,E1 93.212} C_DIS
LIN {X 0.187,Y -564.811,Z 1225.317,A 0.000,B 0.000,C 90.000,E1 93.037} C_DIS
LIN {X 0.175,Y -564.924,Z 1225.313,A 0.000,B 0.000,C 90.000,E1 92.350} C_DIS
LIN {X -0.042,Y -566.349,Z 1225.301,A 0.000,B 0.000,C 90.000,E1 90.172} C_DIS
LIN {X 0.095,Y -567.523,Z 1225.292,A 0.000,B 0.000,C 90.000,E1 88.511} C_DIS
LIN {X -0.152,Y -568.925,Z 1225.281,A 0.000,B 0.000,C 90.000,E1 86.617} C_DIS
LIN {X 0.205,Y -570.497,Z 1225.271,A 0.000,B 0.000,C 90.000,E1 84.666} C_DIS
LIN {X 0.138,Y -572.278,Z 1225.260,A 0.000,B 0.000,C 90.000,E1 82.761} C_DIS
LIN {X -0.198,Y -573.506,Z 1225.252,A 0.000,B 0.000,C 90.000,E1 81.432} C_DIS
LIN {X -0.063,Y -574.431,Z 1225.246,A 0.000,B 0.000,C 90.000,E1 80.330} C_DIS
LIN {X -0.280,Y -575.344,Z 1225.239,A 0.000,B 0.000,C 90.000,E1 78.993} C_DIS
LIN {X -0.163,Y -576.394,Z 1225.230,A 0.000,B 0.000,C 90.000,E1 77.353} C_DIS
LIN {X -0.100,Y -577.187,Z 1225.222,A 0.000,B 0.000,C 90.000,E1 75.992} C_DIS
LIN {X 0.330,Y -577.765,Z 1225.216,A 0.000,B 0.000,C 90.000,E1 74.866} C_DIS
LIN {X 0.071,Y -578.663,Z 1225.207,A 0.000,B 0.000,C 90.000,E1 73.268} C_DIS
LIN {X -0.223,Y -579.405,Z 1225.200,A 0.000,B 0.000,C 90.000,E1 71.945} C_DIS
LIN {X 0.074,Y -580.394,Z 1225.191,A 0.000,B 0.000,C 90.000,E1 70.296} C_DIS
LIN {X 0.301,Y -581.980,Z 1225.177,A 0.000,B 0.000,C 90.000,E1 67.847} C_DIS
LIN {X -0.067,Y -583.141,Z 1225.170,A 0.000,B 0.000,C 90.000,E1 66.538} C_DIS
LIN {X 0.112,Y -584.389,Z 1225.162,A 0.000,B 0.000,C 90.000,E1 65.177} C_DIS
LIN {X -0.083,Y -586.279,Z 1225.150,A 0.000,B 0.000,C 90.000,E1 63.050} C_DIS
LIN {X -0.100,Y -588.218,Z 1225.140,A 0.000,B 0.000,C 90.000,E1 61.179} C_DIS
LIN {X -0.379,Y -589.601,Z 1225.132,A 0.000,B 0.000,C 90.000,E1 59.871} C_DIS
LIN {X -0.342,Y -590.970,Z 1225.125,A 0.000,B 0.000,C 90.000,E1 58.535} C_DIS
LIN {X 0.033,Y -592.186,Z 1225.118,A 0.000,B 0.000,C 90.000,E1 57.168} C_DIS
LIN {X -0.176,Y -593.526,Z 1225.109,A 0.000,B 0.000,C 90.000,E1 55.595} C_DIS
LIN {X -0.127,Y -594.341,Z 1225.103,A 0.000,B 0.000,C 90.000,E1 54.529} C_DIS
LIN {X -0.062,Y -595.216,Z 1225.097,A 0.000,B 0.000,C 90.000,E1 53.463} C_DIS
LIN {X -0.136,Y -596.599,Z 1225.087,A 0.000,B 0.000,C 90.000,E1 51.618} C_DIS
LIN {X 0.086,Y -597.204,Z 1225.082,A 0.000,B 0.000,C 90.000,E1 50.803} C_DIS
LIN {X 0.093,Y -597.891,Z 1225.073,A 0.000,B 0.000,C 90.000,E1 49.218} C_DIS
LIN {X 0.113,Y -598.626,Z 1225.065,A 0.000,B 0.000,C 90.000,E1 47.634} C_DIS
LIN {X 0.315,Y -598.976,Z 1225.057,A 0.000,B 0.000,C 90.000,E1 46.296} C_DIS
LIN {X 0.309,Y -599.052,Z 1225.052,A 0.000,B 0.000,C 90.000,E1 45.243} C_DIS
LIN {X 0.304,Y -598.964,Z 1225.046,A 0.000,B 0.000,C 90.000,E1 44.190} C_DIS
LIN {X -0.117,Y -598.636,Z 1225.040,A 0.000,B 0.000,C 90.000,E1 43.176} C_DIS
LIN {X 0.080,Y -598.311,Z 1225.035,A 0.000,B 0.000,C 90.000,E1 42.366} C_DIS
LIN {X -0.128,Y -597.603,Z 1225.028,A 0.000,B 0.000,C 90.000,E1 41.067} C_DIS
LIN {X -0.125,Y -596.701,Z 1225.019,A 0.000,B 0.000,C 90.000,E1 39.483} C_DIS
LIN {X 0.325,Y -595.849,Z 1225.013,A 0.000,B 0.000,C 90.000,E1 38.382} C_DIS
LIN {X -0.073,Y -594.801,Z 1225.008,A 0.000,B 0.000,C 90.000,E1 37.363} C_DIS
LIN {X -0.013,Y -593.458,Z 1225.002,A 0.000,B 0.000,C 90.000,E1 36.297} C_DIS
LIN {X 0.028,Y -591.900,Z 1224.996,A 0.000,B 0.000,C 90.000,E1 35.231} C_DIS
LIN {X -0.291,Y -589.919,Z 1224.990,A 0.000,B 0.000,C 90.000,E1 34.199} C_DIS
LIN {X -0.013,Y -588.172,Z 1224.985,A 0.000,B 0.000,C 90.000,E1 33.372} C_DIS
LIN {X 0.294,Y -584.652,Z 1224.978,A 0.000,B 0.000,C 90.000,E1 32.005} C_DIS
LIN {X 0.335,Y -582.943,Z 1224.975,A 0.000,B 0.000,C 90.000,E1 31.465} C_DIS
LIN {X 0.365,Y -581.058,Z 1224.972,A 0.000,B 0.000,C 90.000,E1 30.924} C_DIS
LIN {X 0.234,Y -577.877,Z 1224.968,A 0.000,B 0.000,C 90.000,E1 30.129} C_DIS
LIN {X 0.071,Y -574.351,Z 1224.963,A 0.000,B 0.000,C 90.000,E1 29.333} C_DIS
LIN {X -0.162,Y -572.410,Z 1224.961,A 0.000,B 0.000,C 90.000,E1 28.949} C_DIS
LIN {X 0.114,Y -568.051,Z 1224.956,A 0.000,B 0.000,C 90.000,E1 28.103} C_DIS
LIN {X -0.162,Y -563.389,Z 1224.952,A 0.000,B 0.000,C 90.000,E1 27.308} C_DIS
LIN {X -0.045,Y -559.992,Z 1224.949,A 0.000,B 0.000,C 90.000,E1 26.744} C_DIS
LIN {X 0.052,Y -556.372,Z 1224.946,A 0.000,B 0.000,C 90.000,E1 26.181} C_DIS
LIN {X -0.132,Y -552.481,Z 1224.942,A 0.000,B 0.000,C 90.000,E1 25.643} C_DIS
LIN {X 0.028,Y -549.444,Z 1224.940,A 0.000,B 0.000,C 90.000,E1 25.207} C_DIS
LIN {X 0.235,Y -541.611,Z 1224.935,A 0.000,B 0.000,C 90.000,E1 24.207} C_DIS
LIN {X -0.009,Y -534.341,Z 1224.930,A 0.000,B 0.000,C 90.000,E1 23.387} C_DIS
LIN {X 0.059,Y -530.497,Z 1224.928,A 0.000,B 0.000,C 90.000,E1 22.950} C_DIS
LIN {X 0.073,Y -521.443,Z 1224.922,A 0.000,B 0.000,C 90.000,E1 21.972} C_DIS
LIN {X -0.189,Y -512.152,Z 1224.917,A 0.000,B 0.000,C 90.000,E1 21.046} C_DIS
LIN {X -0.129,Y -500.954,Z 1224.911,A 0.000,B 0.000,C 90.000,E1 19.939} C_DIS
LIN {X 0.153,Y -490.888,Z 1224.906,A 0.000,B 0.000,C 90.000,E1 18.960} C_DIS
LIN {X 0.057,Y -483.582,Z 1224.902,A 0.000,B 0.000,C 90.000,E1 18.308} C_DIS
LIN {X -0.136,Y -470.175,Z 1224.895,A 0.000,B 0.000,C 90.000,E1 17.149} C_DIS
LIN {X -0.120,Y -456.997,Z 1224.889,A 0.000,B 0.000,C 90.000,E1 15.969} C_DIS
LIN {X -0.248,Y -440.852,Z 1224.880,A 0.000,B 0.000,C 90.000,E1 14.481} C_DIS
LIN {X 0.107,Y -422.123,Z 1224.870,A 0.000,B 0.000,C 90.000,E1 12.535} C_DIS
LIN {X -0.035,Y -404.236,Z 1224.859,A 0.000,B 0.000,C 90.000,E1 10.546} C_DIS
LIN {X 0.124,Y -398.100,Z 1224.854,A 0.000,B 0.000,C 90.000,E1 9.726} C_DIS
LIN {X 0.153,Y -394.880,Z 1224.851,A 0.000,B 0.000,C 90.000,E1 9.208} C_DIS
LIN {X -0.048,Y -393.951,Z 1224.850,A 0.000,B 0.000,C 90.000,E1 8.973} C_DIS
LIN {X -0.086,Y -393.949,Z 1224.850,A 0.000,B 0.000,C 90.000,E1 8.973} C_DIS
LIN {X 0.096,Y -394.025,Z 1224.848,A 0.000,B 0.000,C 90.000,E1 8.681} C_DIS
LIN {X 0.058,Y -394.034,Z 1224.848,A 0.000,B 0.000,C 90.000,E1 8.681} C_DIS
LIN {X -0.171,Y -396.727,Z 1224.845,A 0.000,B 0.000,C 90.000,E1 8.106} C_DIS
LIN {X -0.132,Y -400.043,Z 1224.843,A 0.000,B 0.000,C 90.000,E1 7.701} C_DIS
LIN {X 0.208,Y -403.346,Z 1224.841,A 0.000,B 0.000,C 90.000,E1 7.352} C_DIS
LIN {X -0.042,Y -419.742,Z 1224.834,A 0.000,B 0.000,C 90.000,E1 6.144} C_DIS
LIN {X -0.022,Y -434.138,Z 1224.828,A 0.000,B 0.000,C 90.000,E1 5.049} C_DIS
LIN {X -0.040,Y -446.803,Z 1224.823,A 0.000,B 0.000,C 90.000,E1 4.073} C_DIS
LIN {X 0.152,Y -459.267,Z 1224.817,A 0.000,B 0.000,C 90.000,E1 3.094} C_DIS
LIN {X -0.217,Y -468.512,Z 1224.813,A 0.000,B 0.000,C 90.000,E1 2.407} C_DIS
LIN {X 0.011,Y -472.997,Z 1224.811,A 0.000,B 0.000,C 90.000,E1 2.007} C_DIS
LIN {X -0.006,Y -478.862,Z 1224.808,A 0.000,B 0.000,C 90.000,E1 1.489} C_DIS
LIN {X -0.146,Y -485.667,Z 1224.805,A 0.000,B 0.000,C 90.000,E1 0.859} C_DIS
LIN {X -0.216,Y -492.448,Z 1224.801,A 0.000,B 0.000,C 90.000,E1 0.172} C_DIS
LIN {X 0.130,Y -498.323,Z 1224.797,A 0.000,B 0.000,C 90.000,E1 359.484} C_DIS
LIN {X -0.214,Y -504.410,Z 1224.793,A 0.000,B 0.000,C 90.000,E1 358.797} C_DIS
LIN {X -0.201,Y -510.150,Z 1224.789,A 0.000,B 0.000,C 90.000,E1 358.051} C_DIS
LIN {X -0.165,Y -515.400,Z 1224.785,A 0.000,B 0.000,C 90.000,E1 357.306} C_DIS
LIN {X -0.059,Y -520.316,Z 1224.781,A 0.000,B 0.000,C 90.000,E1 356.560} C_DIS
LIN {X -0.175,Y -523.988,Z 1224.778,A 0.000,B 0.000,C 90.000,E1 355.988} C_DIS
LIN {X 0.013,Y -528.144,Z 1224.774,A 0.000,B 0.000,C 90.000,E1 355.241} C_DIS
LIN {X -0.009,Y -531.207,Z 1224.770,A 0.000,B 0.000,C 90.000,E1 354.666} C_DIS
LIN {X 0.027,Y -535.331,Z 1224.766,A 0.000,B 0.000,C 90.000,E1 353.799} C_DIS
LIN {X -0.203,Y -537.270,Z 1224.763,A 0.000,B 0.000,C 90.000,E1 353.394} C_DIS
LIN {X -0.096,Y -540.762,Z 1224.758,A 0.000,B 0.000,C 90.000,E1 352.527} C_DIS
LIN {X -0.031,Y -542.951,Z 1224.755,A 0.000,B 0.000,C 90.000,E1 351.951} C_DIS
LIN {X 0.133,Y -545.943,Z 1224.751,A 0.000,B 0.000,C 90.000,E1 351.084} C_DIS
LIN {X -0.216,Y -548.626,Z 1224.746,A 0.000,B 0.000,C 90.000,E1 350.274} C_DIS
LIN {X 0.208,Y -551.822,Z 1224.740,A 0.000,B 0.000,C 90.000,E1 349.106} C_DIS
LIN {X 0.269,Y -555.471,Z 1224.732,A 0.000,B 0.000,C 90.000,E1 347.701} C_DIS
LIN {X 0.119,Y -557.404,Z 1224.727,A 0.000,B 0.000,C 90.000,E1 346.881} C_DIS
LIN {X -0.140,Y -560.350,Z 1224.719,A 0.000,B 0.000,C 90.000,E1 345.519} C_DIS
LIN {X 0.046,Y -562.539,Z 1224.713,A 0.000,B 0.000,C 90.000,E1 344.393} C_DIS
LIN {X -0.283,Y -564.493,Z 1224.707,A 0.000,B 0.000,C 90.000,E1 343.323} C_DIS
LIN {X 0.117,Y -566.210,Z 1224.701,A 0.000,B 0.000,C 90.000,E1 342.181} C_DIS
LIN {X 0.340,Y -568.029,Z 1224.693,A 0.000,B 0.000,C 90.000,E1 340.786} C_DIS
LIN {X -0.093,Y -568.961,Z 1224.689,A 0.000,B 0.000,C 90.000,E1 340.007} C_DIS
LIN {X -0.326,Y -569.610,Z 1224.684,A 0.000,B 0.000,C 90.000,E1 339.209} C_DIS
LIN {X 0.189,Y -570.057,Z 1224.680,A 0.000,B 0.000,C 90.000,E1 338.337} C_DIS
LIN {X -0.029,Y -570.259,Z 1224.675,A 0.000,B 0.000,C 90.000,E1 337.539} C_DIS
LIN {X -0.077,Y -569.770,Z 1224.668,A 0.000,B 0.000,C 90.000,E1 336.177} C_DIS
LIN {X -0.080,Y -568.978,Z 1224.663,A 0.000,B 0.000,C 90.000,E1 335.357} C_DIS
LIN {X -0.089,Y -567.967,Z 1224.659,A 0.000,B 0.000,C 90.000,E1 334.537} C_DIS
LIN {X 0.067,Y -567.030,Z 1224.656,A 0.000,B 0.000,C 90.000,E1 333.973} C_DIS
LIN {X 0.285,Y -565.316,Z 1224.651,A 0.000,B 0.000,C 90.000,E1 333.127} C_DIS
LIN {X 0.299,Y -562.526,Z 1224.645,A 0.000,B 0.000,C 90.000,E1 332.025} C_DIS
LIN {X -0.288,Y -559.974,Z 1224.640,A 0.000,B 0.000,C 90.000,E1 331.257} C_DIS
LIN {X 0.130,Y -556.506,Z 1224.636,A 0.000,B 0.000,C 90.000,E1 330.383} C_DIS
LIN {X -0.302,Y -553.924,Z 1224.632,A 0.000,B 0.000,C 90.000,E1 329.871} C_DIS
LIN {X 0.047,Y -549.274,Z 1224.628,A 0.000,B 0.000,C 90.000,E1 328.997} C_DIS
LIN {X -0.156,Y -545.849,Z 1224.625,A 0.000,B 0.000,C 90.000,E1 328.456} C_DIS
LIN {X -0.054,Y -541.140,Z 1224.621,A 0.000,B 0.000,C 90.000,E1 327.740} C_DIS
LIN {X -0.173,Y -538.157,Z 1224.618,A 0.000,B 0.000,C 90.000,E1 327.327} C_DIS
LIN {X 0.114,Y -528.110,Z 1224.611,A 0.000,B 0.000,C 90.000,E1 326.008} C_DIS
LIN {X 0.055,Y -516.799,Z 1224.603,A 0.000,B 0.000,C 90.000,E1 324.562} C_DIS
LIN {X 0.112,Y -513.966,Z 1224.601,A 0.000,B 0.000,C 90.000,E1 324.116} C_DIS
LIN {X -0.030,Y -511.193,Z 1224.598,A 0.000,B 0.000,C 90.000,E1 323.623} C_DIS
LIN {X 0.265,Y -509.582,Z 1224.595,A 0.000,B 0.000,C 90.000,E1 323.130} C_DIS
LIN {X 0.069,Y -509.180,Z 1224.595,A 0.000,B 0.000,C 90.000,E1 323.004} C_DIS
LIN {X -0.003,Y -507.824,Z 1224.590,A 0.000,B 0.000,C 90.000,E1 322.271} C_DIS
LIN {X 0.143,Y -507.285,Z 1224.586,A 0.000,B 0.000,C 90.000,E1 321.376} C_DIS
LIN {X -0.155,Y -507.275,Z 1224.581,A 0.000,B 0.000,C 90.000,E1 320.517} C_DIS
LIN {X 0.015,Y -508.645,Z 1224.567,A 0.000,B 0.000,C 90.000,E1 318.119} C_DIS
LIN {X 0.144,Y -509.467,Z 1224.559,A 0.000,B 0.000,C 90.000,E1 316.620} C_DIS
LIN {X -0.073,Y -510.168,Z 1224.551,A 0.000,B 0.000,C 90.000,E1 315.162} C_DIS
LIN {X -0.129,Y -511.036,Z 1224.539,A 0.000,B 0.000,C 90.000,E1 313.095} C_DIS
LIN {X -0.041,Y -511.842,Z 1224.530,A 0.000,B 0.000,C 90.000,E1 311.310} C_DIS
LIN {X 0.280,Y -512.378,Z 1224.523,A 0.000,B 0.000,C 90.000,E1 310.092} C_DIS
LIN {X -0.120,Y -512.825,Z 1224.516,A 0.000,B 0.000,C 90.000,E1 308.955} C_DIS
LIN {X 0.051,Y -513.436,Z 1224.505,A 0.000,B 0.000,C 90.000,E1 306.870} C_DIS
LIN {X 0.089,Y -513.950,Z 1224.497,A 0.000,B 0.000,C 90.000,E1 305.391} C_DIS
LIN {X 0.058,Y -514.539,Z 1224.487,A 0.000,B 0.000,C 90.000,E1 303.627} C_DIS
LIN {X -0.105,Y -514.893,Z 1224.480,A 0.000,B 0.000,C 90.000,E1 302.467} C_DIS
LIN {X 0.173,Y -515.102,Z 1224.474,A 0.000,B 0.000,C 90.000,E1 301.258} C_DIS
LIN {X -0.239,Y -515.333,Z 1224.464,A 0.000,B 0.000,C 90.000,E1 299.539} C_DIS
LIN {X -0.210,Y -515.429,Z 1224.458,A 0.000,B 0.000,C 90.000,E1 298.359} C_DIS
LIN {X 0.273,Y -515.562,Z 1224.451,A 0.000,B 0.000,C 90.000,E1 297.129} C_DIS
LIN {X 0.192,Y -515.617,Z 1224.439,A 0.000,B 0.000,C 90.000,E1 295.079} C_DIS
LIN {X -0.110,Y -515.759,Z 1224.431,A 0.000,B 0.000,C 90.000,E1 293.643} C_DIS
LIN {X 0.069,Y -515.758,Z 1224.423,A 0.000,B 0.000,C 90.000,E1 292.153} C_DIS
LIN {X 0.239,Y -515.349,Z 1224.415,A 0.000,B 0.000,C 90.000,E1 290.663} C_DIS
LIN {X 0.086,Y -514.733,Z 1224.408,A 0.000,B 0.000,C 90.000,E1 289.504} C_DIS
LIN {X -0.164,Y -513.935,Z 1224.399,A 0.000,B 0.000,C 90.000,E1 287.764} C_DIS
LIN {X 0.106,Y -513.196,Z 1224.391,A 0.000,B 0.000,C 90.000,E1 286.260} C_DIS
LIN {X 0.247,Y -512.663,Z 1224.384,A 0.000,B 0.000,C 90.000,E1 285.064} C_DIS
LIN {X 0.145,Y -511.403,Z 1224.372,A 0.000,B 0.000,C 90.000,E1 283.008} C_DIS
LIN {X 0.087,Y -510.395,Z 1224.364,A 0.000,B 0.000,C 90.000,E1 281.535} C_DIS
LIN {X -0.023,Y -509.775,Z 1224.359,A 0.000,B 0.000,C 90.000,E1 280.658} C_DIS
LIN {X 0.103,Y -508.311,Z 1224.348,A 0.000,B 0.000,C 90.000,E1 278.568} C_DIS
LIN {X 0.113,Y -506.963,Z 1224.336,A 0.000,B 0.000,C 90.000,E1 276.486} C_DIS
LIN {X -0.204,Y -505.514,Z 1224.321,A 0.000,B 0.000,C 90.000,E1 273.841} C_DIS
LIN {X -0.104,Y -504.775,Z 1224.315,A 0.000,B 0.000,C 90.000,E1 272.636} C_DIS
LIN {X -0.018,Y -503.978,Z 1224.308,A 0.000,B 0.000,C 90.000,E1 271.432} C_DIS
LIN {X 0.212,Y -502.655,Z 1224.296,A 0.000,B 0.000,C 90.000,E1 269.312} C_DIS
LIN {X -0.233,Y -501.957,Z 1224.290,A 0.000,B 0.000,C 90.000,E1 268.165} C_DIS
LIN {X 0.077,Y -500.983,Z 1224.280,A 0.000,B 0.000,C 90.000,E1 266.331} C_DIS
LIN {X 0.013,Y -499.944,Z 1224.271,A 0.000,B 0.000,C 90.000,E1 264.837} C_DIS
LIN {X 0.065,Y -499.116,Z 1224.265,A 0.000,B 0.000,C 90.000,E1 263.628} C_DIS
LIN {X 0.162,Y -498.034,Z 1224.258,A 0.000,B 0.000,C 90.000,E1 262.413} C_DIS
LIN {X -0.180,Y -495.852,Z 1224.245,A 0.000,B 0.000,C 90.000,E1 260.038} C_DIS
LIN {X -0.049,Y -494.758,Z 1224.238,A 0.000,B 0.000,C 90.000,E1 258.814} C_DIS
LIN {X 0.159,Y -492.658,Z 1224.223,A 0.000,B 0.000,C 90.000,E1 256.061} C_DIS
LIN {X -0.095,Y -491.436,Z 1224.213,A 0.000,B 0.000,C 90.000,E1 254.267} C_DIS
LIN {X 0.012,Y -490.166,Z 1224.199,A 0.000,B 0.000,C 90.000,E1 251.819} C_DIS
LIN {X -0.003,Y -489.429,Z 1224.191,A 0.000,B 0.000,C 90.000,E1 250.296} C_DIS
LIN {X -0.060,Y -488.813,Z 1224.184,A 0.000,B 0.000,C 90.000,E1 249.082} C_DIS
LIN {X 0.047,Y -488.186,Z 1224.177,A 0.000,B 0.000,C 90.000,E1 247.847} C_DIS
LIN {X 0.159,Y -487.083,Z 1224.168,A 0.000,B 0.000,C 90.000,E1 246.305} C_DIS
LIN {X 0.213,Y -485.535,Z 1224.158,A 0.000,B 0.000,C 90.000,E1 244.460} C_DIS
LIN {X 0.016,Y -484.315,Z 1224.151,A 0.000,B 0.000,C 90.000,E1 243.256} C_DIS
LIN {X 0.018,Y -483.199,Z 1224.145,A 0.000,B 0.000,C 90.000,E1 242.025} C_DIS
LIN {X 0.002,Y -481.896,Z 1224.138,A 0.000,B 0.000,C 90.000,E1 240.795} C_DIS
LIN {X 0.197,Y -480.446,Z 1224.131,A 0.000,B 0.000,C 90.000,E1 239.537} C_DIS
LIN {X 0.163,Y -478.747,Z 1224.122,A 0.000,B 0.000,C 90.000,E1 237.995} C_DIS
LIN {X -0.116,Y -476.587,Z 1224.112,A 0.000,B 0.000,C 90.000,E1 236.167} C_DIS
LIN {X -0.127,Y -474.183,Z 1224.100,A 0.000,B 0.000,C 90.000,E1 233.989} C_DIS
LIN {X 0.138,Y -472.524,Z 1224.091,A 0.000,B 0.000,C 90.000,E1 232.396} C_DIS
LIN {X -0.004,Y -470.159,Z 1224.077,A 0.000,B 0.000,C 90.000,E1 229.908} C_DIS
LIN {X 0.115,Y -468.812,Z 1224.069,A 0.000,B 0.000,C 90.000,E1 228.324} C_DIS
LIN {X -0.003,Y -466.842,Z 1224.056,A 0.000,B 0.000,C 90.000,E1 226.134} C_DIS
LIN {X -0.011,Y -465.020,Z 1224.000,A 0.000,B 0.000,C 90.000,E1 216.011} C_DIS
LIN {X -0.225,Y -468.730,Z 1223.970,A 0.000,B 0.000,C 90.000,E1 210.669} C_DIS
LIN {X -0.100,Y -472.138,Z 1223.953,A 0.000,B 0.000,C 90.000,E1 207.513} C_DIS
LIN {X -0.189,Y -474.821,Z 1223.941,A 0.000,B 0.000,C 90.000,E1 205.335} C_DIS
LIN {X -0.053,Y -480.457,Z 1223.920,A 0.000,B 0.000,C 90.000,E1 201.589} C_DIS
LIN {X 0.086,Y -486.343,Z 1223.903,A 0.000,B 0.000,C 90.000,E1 198.489} C_DIS
LIN {X -0.141,Y -489.707,Z 1223.894,A 0.000,B 0.000,C 90.000,E1 196.985} C_DIS
LIN {X 0.080,Y -494.874,Z 1223.882,A 0.000,B 0.000,C 90.000,E1 194.828} C_DIS
LIN {X 0.222,Y -498.849,Z 1223.874,A 0.000,B 0.000,C 90.000,E1 193.300} C_DIS
LIN {X -0.045,Y -502.948,Z 1223.866,A 0.000,B 0.000,C 90.000,E1 191.827} C_DIS
LIN {X 0.095,Y -507.889,Z 1223.856,A 0.000,B 0.000,C 90.000,E1 190.018} C_DIS
LIN {X -0.209,Y -512.256,Z 1223.848,A 0.000,B 0.000,C 90.000,E1 188.568} C_DIS
LIN {X 0.097,Y -515.748,Z 1223.841,A 0.000,B 0.000,C 90.000,E1 187.352} C_DIS
LIN {X -0.137,Y -520.035,Z 1223.833,A 0.000,B 0.000,C 90.000,E1 185.910} C_DIS
LIN {X 0.119,Y -525.905,Z 1223.821,A 0.000,B 0.000,C 90.000,E1 183.841} C_DIS
LIN {X -0.034,Y -531.024,Z 1223.812,A 0.000,B 0.000,C 90.000,E1 182.121} C_DIS
LIN {X -0.076,Y -536.017,Z 1223.802,A 0.000,B 0.000,C 90.000,E1 180.401} C_DIS
LIN {X -0.037,Y -540.120,Z 1223.794,A 0.000,B 0.000,C 90.000,E1 178.969} C_DIS
LIN {X 0.088,Y -544.133,Z 1223.786,A 0.000,B 0.000,C 90.000,E1 177.535} C_DIS
LIN {X -0.262,Y -547.917,Z 1223.779,A 0.000,B 0.000,C 90.000,E1 176.159} C_DIS
LIN {X 0.033,Y -551.568,Z 1223.771,A 0.000,B 0.000,C 90.000,E1 174.723} C_DIS
LIN {X -0.210,Y -554.425,Z 1223.765,A 0.000,B 0.000,C 90.000,E1 173.628} C_DIS
LIN {X -0.158,Y -558.581,Z 1223.755,A 0.000,B 0.000,C 90.000,E1 171.951} C_DIS
LIN {X -0.019,Y -562.670,Z 1223.746,A 0.000,B 0.000,C 90.000,E1 170.274} C_DIS
LIN {X 0.232,Y -566.012,Z 1223.738,A 0.000,B 0.000,C 90.000,E1 168.870} C_DIS
LIN {X -0.007,Y -571.395,Z 1223.726,A 0.000,B 0.000,C 90.000,E1 166.700} C_DIS
LIN {X -0.173,Y -576.316,Z 1223.716,A 0.000,B 0.000,C 90.000,E1 164.810} C_DIS
LIN {X -0.310,Y -585.516,Z 1223.698,A 0.000,B 0.000,C 90.000,E1 161.583} C_DIS
LIN {X -0.150,Y -597.653,Z 1223.678,A 0.000,B 0.000,C 90.000,E1 158.103} C_DIS
LIN {X -0.171,Y -601.788,Z 1223.672,A 0.000,B 0.000,C 90.000,E1 157.050} C_DIS
LIN {X -0.256,Y -607.877,Z 1223.664,A 0.000,B 0.000,C 90.000,E1 155.485} C_DIS
LIN {X 0.112,Y -611.806,Z 1223.658,A 0.000,B 0.000,C 90.000,E1 154.409} C_DIS
LIN {X -0.039,Y -616.596,Z 1223.651,A 0.000,B 0.000,C 90.000,E1 153.127} C_DIS
LIN {X -0.115,Y -621.106,Z 1223.644,A 0.000,B 0.000,C 90.000,E1 151.847} C_DIS
LIN {X 0.174,Y -625.490,Z 1223.636,A 0.000,B 0.000,C 90.000,E1 150.539} C_DIS
LIN {X 0.333,Y -630.708,Z 1223.628,A 0.000,B 0.000,C 90.000,E1 148.997} C_DIS
LIN {X -0.299,Y -634.852,Z 1223.621,A 0.000,B 0.000,C 90.000,E1 147.788} C_DIS
LIN {X -0.026,Y -638.034,Z 1223.615,A 0.000,B 0.000,C 90.000,E1 146.755} C_DIS
LIN {X -0.197,Y -641.768,Z 1223.608,A 0.000,B 0.000,C 90.000,E1 145.515} C_DIS
LIN {X 0.246,Y -643.155,Z 1223.606,A 0.000,B 0.000,C 90.000,E1 144.975} C_DIS
LIN {X 0.000,Y -646.434,Z 1223.599,A 0.000,B 0.000,C 90.000,E1 143.749} C_DIS
LIN {X -0.013,Y -648.215,Z 1223.594,A 0.000,B 0.000,C 90.000,E1 143.004} C_DIS
LIN {X 0.222,Y -651.132,Z 1223.588,A 0.000,B 0.000,C 90.000,E1 141.743} C_DIS
LIN {X -0.343,Y -653.402,Z 1223.582,A 0.000,B 0.000,C 90.000,E1 140.803} C_DIS
LIN {X -0.016,Y -656.126,Z 1223.575,A 0.000,B 0.000,C 90.000,E1 139.542} C_DIS
LIN {X -0.203,Y -659.949,Z 1223.566,A 0.000,B 0.000,C 90.000,E1 137.838} C_DIS
LIN {X -0.287,Y -663.155,Z 1223.558,A 0.000,B 0.000,C 90.000,E1 136.377} C_DIS
LIN {X -0.334,Y -668.337,Z 1223.545,A 0.000,B 0.000,C 90.000,E1 134.190} C_DIS
LIN {X 0.218,Y -672.630,Z 1223.536,A 0.000,B 0.000,C 90.000,E1 132.447} C_DIS
